  Call Extruder(264.21579)
  MoveL 9606 to (525.09, 528.57, 172) mm, rotated rx 180 ry 0 rz 160 deg; joints [9.282, 56.814, -9.011, -142.877, 54.137, 156.086]
  Call Extruder(269.11621)
  MoveL 9607 to (523.93, 529.55, 172) mm, rotated rx -180 ry 0 rz 160 deg; joints [9.42, 56.63, -8.662, -142.793, 54.323, 156.117]
  Set speed (17.5 mm/s)
  Call Extruder(272.14590)
  MoveL 9608 to (523.2, 530.13, 172) mm, rotated rx -180 ry 0 rz 160 deg; joints [9.503, 56.512, -8.44, -142.745, 54.44, 156.14]
  Set speed (17.5 mm/s)
  Call Extruder(276.64119)
  MoveL 9609 to (522.08, 530.96, 172) mm, rotated rx -180 ry 0 rz 160 deg; joints [9.623, 56.332, -8.101, -142.679, 54.616, 156.181]
  Set speed (17.5 mm/s)
  Call Extruder(279.35040)
  MoveL 9610 to (521.39, 531.44, 172) mm, rotated rx 180 ry 0 rz 160 deg; joints [9.693, 56.221, -7.89, -142.643, 54.723, 156.208]
  Set speed (17.5 mm/s)
  Call Extruder(281.76760)
  MoveL 9611 to (520.77, 531.85, 172) mm, rotated rx -180 ry 0 rz 160 deg; joints [9.755, 56.12, -7.7, -142.612, 54.819, 156.235]
  Set speed (17.5 mm/s)
  Call Extruder(284.79201)
  MoveL 9612 to (519.98, 532.36, 172) mm, rotated rx 180 ry 0 rz 160 deg; joints [9.831, 55.992, -7.459, -142.576, 54.939, 156.27]
  Set speed (17.5 mm/s)
  Call Extruder(286.82384)
  MoveL 9613 to (519.44, 532.68, 172) mm, rotated rx 180 ry 0 rz 160 deg; joints [9.881, 55.905, -7.294, -142.553, 55.021, 156.296]
  Set speed (17.5 mm/s)
  Call Extruder(289.33819)
  MoveL 9614 to (518.77, 533.08, 172) mm, rotated rx 180 ry 0 rz 160 deg; joints [9.941, 55.795, -7.088, -142.527, 55.122, 156.329]
  Set speed (17.5 mm/s)
  Call Extruder(291.88729)
  MoveL 9615 to (518.08, 533.46, 172) mm, rotated rx 180 ry 0 rz 160 deg; joints [10.001, 55.682, -6.875, -142.502, 55.225, 156.365]
  Call Extruder(294.64849)
  MoveL 9616 to (517.32, 533.86, 172) mm, rotated rx 180 ry 0 rz 160 deg; joints [10.064, 55.559, -6.642, -142.478, 55.337, 156.406]
  Set speed (17.5 mm/s)
  Call Extruder(299.60980)
  MoveL 9617 to (515.94, 534.53, 172) mm, rotated rx -180 ry 0 rz 160 deg; joints [10.173, 55.333, -6.215, -142.44, 55.54, 156.485]
  Set speed (17.5 mm/s)
  Call Extruder(304.71552)
  MoveL 9618 to (514.49, 535.16, 172) mm, rotated rx 180 ry 0 rz 160 deg; joints [10.28, 55.095, -5.766, -142.41, 55.75, 156.574]
  Set speed (17.5 mm/s)
  Call Extruder(309.41983)
  MoveL 9619 to (513.13, 535.69, 172) mm, rotated rx -180 ry 0 rz 160 deg; joints [10.373, 54.871, -5.344, -142.388, 55.944, 156.662]
  Call Extruder(314.52276)
  MoveL 9620 to (511.64, 536.2, 172) mm, rotated rx -180 ry 0 rz 160 deg; joints [10.468, 54.624, -4.879, -142.373, 56.154, 156.765]
  Set speed (17.5 mm/s)
  Call Extruder(319.40100)
  MoveL 9621 to (510.19, 536.64, 172) mm, rotated rx 180 ry 0 rz 160 deg; joints [10.553, 54.384, -4.427, -142.366, 56.356, 156.869]
  Set speed (17.5 mm/s)
  Call Extruder(324.41187)
  MoveL 9622 to (508.69, 537.02, 172) mm, rotated rx 180 ry 0 rz 160 deg; joints [10.633, 54.135, -3.957, -142.367, 56.562, 156.981]
  Set speed (17.5 mm/s)
  Call Extruder(329.43968)
  MoveL 9623 to (507.17, 537.35, 172) mm, rotated rx 180 ry 0 rz 160 deg; joints [10.707, 53.882, -3.479, -142.376, 56.768, 157.1]
  Set speed (17.5 mm/s)
  Call Extruder(334.69209)
  MoveL 9624 to (505.57, 537.62, 172) mm, rotated rx -180 ry 0 rz 160 deg; joints [10.777, 53.614, -2.975, -142.393, 56.983, 157.231]
  Call Extruder(339.62073)
  MoveL 9625 to (504.05, 537.81, 172) mm, rotated rx -180 ry 0 rz 160 deg; joints [10.835, 53.361, -2.498, -142.417, 57.183, 157.359]
  Set speed (17.5 mm/s)
  Call Extruder(344.69311)
  MoveL 9626 to (502.49, 537.95, 172) mm, rotated rx 180 ry 0 rz 160 deg; joints [10.889, 53.099, -2.004, -142.449, 57.387, 157.495]
  Call Extruder(349.77465)
  MoveL 9627 to (500.91, 538.02, 172) mm, rotated rx -180 ry 0 rz 160 deg; joints [10.934, 52.835, -1.506, -142.49, 57.59, 157.637]
  Set speed (17.5 mm/s)
  Call Extruder(354.61934)
  MoveL 9628 to (499.41, 538.02, 172) mm, rotated rx -180 ry 0 rz 160 deg; joints [10.971, 52.582, -1.03, -142.536, 57.781, 157.776]
  Set speed (10.0 mm/s)
  MoveL 9629 to (499.41, 538.02, 176) mm, rotated rx 180 ry 0 rz 160 deg; joints [10.971, 52.04, -0.954, -142.356, 57.412, 157.44]
  Set speed (120.0 mm/s)
  MoveL 9630 to (499.43, 537.08, 176) mm, rotated rx 180 ry 0 rz 160 deg; joints [10.855, 52.012, -0.902, -142.492, 57.387, 157.526]
  Set speed (17.6 mm/s)
  Call Extruder(359.63179)
  MoveL 9631 to (497.87, 537.03, 176) mm, rotated rx -180 ry 0 rz 160 deg; joints [10.885, 51.747, -0.406, -142.549, 57.581, 157.675]
  Call Extruder(364.52764)
  MoveL 9632 to (496.35, 536.91, 176) mm, rotated rx -180 ry 0 rz 160 deg; joints [10.906, 51.489, 0.078, -142.613, 57.768, 157.825]
  Call Extruder(369.33210)
  MoveL 9633 to (494.87, 536.73, 176) mm, rotated rx 180 ry 0 rz 160 deg; joints [10.92, 51.235, 0.552, -142.682, 57.949, 157.975]
  Set speed (17.6 mm/s)
  Call Extruder(374.09373)
  MoveL 9634 to (493.4, 536.49, 176) mm, rotated rx 180 ry 0 rz 160 deg; joints [10.925, 50.984, 1.022, -142.758, 58.125, 158.128]
  Call Extruder(378.49274)
  MoveL 9635 to (492.06, 536.23, 176) mm, rotated rx -180 ry 0 rz 160 deg; joints [10.925, 50.754, 1.453, -142.834, 58.284, 158.271]
  Set speed (17.6 mm/s)
  Call Extruder(381.55349)
  MoveL 9636 to (491.13, 536.01, 176) mm, rotated rx -180 ry 0 rz 160 deg; joints [10.92, 50.594, 1.751, -142.891, 58.393, 158.372]
  Call Extruder(383.93419)
  MoveL 9637 to (490.41, 535.83, 176) mm, rotated rx -180 ry 0 rz 160 deg; joints [10.914, 50.47, 1.983, -142.937, 58.477, 158.451]
  Set speed (17.6 mm/s)
  Call Extruder(388.87401)
  MoveL 9638 to (488.93, 535.4, 176) mm, rotated rx 180 ry 0 rz 160 deg; joints [10.896, 50.215, 2.46, -143.038, 58.648, 158.618]
  Set speed (17.6 mm/s)
  Call Extruder(393.64536)
  MoveL 9639 to (487.52, 534.93, 176) mm, rotated rx -180 ry 0 rz 160 deg; joints [10.871, 49.971, 2.916, -143.144, 58.808, 158.782]
  Set speed (17.6 mm/s)
  Call Extruder(398.69949)
  MoveL 9640 to (486.06, 534.37, 176) mm, rotated rx -180 ry 0 rz 160 deg; joints [10.835, 49.715, 3.395, -143.262, 58.973, 158.957]
  Set speed (17.6 mm/s)
  Call Extruder(403.34117)
  MoveL 9641 to (484.73, 533.8, 176) mm, rotated rx 180 ry 0 rz 160 deg; joints [10.795, 49.483, 3.828, -143.378, 59.121, 159.12]
  Set speed (17.6 mm/s)
  Call Extruder(407.92857)
  MoveL 9642 to (483.44, 533.18, 176) mm, rotated rx 180 ry 0 rz 160 deg; joints [10.748, 49.256, 4.251, -143.499, 59.262, 159.282]
  Set speed (17.6 mm/s)
  Call Extruder(411.24892)
  MoveL 9643 to (482.52, 532.71, 176) mm, rotated rx -180 ry 0 rz 160 deg; joints [10.71, 49.094, 4.553, -143.59, 59.361, 159.4]
  Set speed (17.6 mm/s)
  Call Extruder(415.20714)
  MoveL 9644 to (481.44, 532.11, 176) mm, rotated rx 180 ry 0 rz 160 deg; joints [10.659, 48.904, 4.908, -143.704, 59.476, 159.542]
  Set speed (17.6 mm/s)
  Call Extruder(417.70243)
  MoveL 9645 to (480.77, 531.71, 176) mm, rotated rx 180 ry 0 rz 160 deg; joints [10.624, 48.786, 5.129, -143.777, 59.546, 159.632]
  Set speed (17.6 mm/s)
  Call Extruder(420.49475)
  MoveL 9646 to (480.03, 531.25, 176) mm, rotated rx 180 ry 0 rz 160 deg; joints [10.583, 48.655, 5.374, -143.862, 59.624, 159.733]
  Call Extruder(425.15951)
  MoveL 9647 to (478.82, 530.45, 176) mm, rotated rx -180 ry 0 rz 160 deg; joints [10.508, 48.439, 5.776, -144.007, 59.749, 159.901]
  Set speed (17.6 mm/s)
  Call Extruder(427.37809)
  MoveL 9648 to (478.26, 530.05, 176) mm, rotated rx 180 ry 0 rz 160 deg; joints [10.469, 48.338, 5.964, -144.079, 59.806, 159.981]
  Set speed (17.6 mm/s)
  Call Extruder(430.26889)
  MoveL 9649 to (477.54, 529.51, 176) mm, rotated rx 180 ry 0 rz 160 deg; joints [10.417, 48.208, 6.207, -144.174, 59.88, 160.086]
  Set speed (17.6 mm/s)
  Call Extruder(432.68875)
  MoveL 9650 to (476.94, 529.05, 176) mm, rotated rx 180 ry 0 rz 160 deg; joints [10.371, 48.101, 6.406, -144.255, 59.939, 160.174]
  Set speed (17.6 mm/s)
  Call Extruder(437.16751)
  MoveL 9651 to (475.87, 528.16, 176) mm, rotated rx 180 ry 0 rz 160 deg; joints [10.281, 47.906, 6.769, -144.41, 60.045, 160.336]
  Set speed (17.6 mm/s)
  Call Extruder(439.64918)
  MoveL 9652 to (475.28, 527.65, 176) mm, rotated rx 180 ry 0 rz 160 deg; joints [10.228, 47.801, 6.967, -144.498, 60.102, 160.426]
  Set speed (17.6 mm/s)
  Call Extruder(443.32920)
  MoveL 9653 to (474.44, 526.87, 176) mm, rotated rx 180 ry 0 rz 160 deg; joints [10.147, 47.647, 7.254, -144.631, 60.183, 160.559]
  Set speed (17.6 mm/s)
  Call Extruder(448.58769)
  MoveL 9654 to (473.28, 525.72, 176) mm, rotated rx 180 ry 0 rz 160 deg; joints [10.022, 47.433, 7.652, -144.827, 60.293, 160.749]
  Set speed (17.6 mm/s)
  Call Extruder(452.04675)
  MoveL 9655 to (472.54, 524.93, 176) mm, rotated rx -180 ry 0 rz 160 deg; joints [9.936, 47.297, 7.905, -144.96, 60.36, 160.873]
  Set speed (17.6 mm/s)
  Call Extruder(457.05308)
  MoveL 9656 to (471.52, 523.76, 176) mm, rotated rx 180 ry 0 rz 160 deg; joints [9.804, 47.106, 8.261, -145.157, 60.452, 161.053]
  Set speed (17.6 mm/s)
  Call Extruder(459.37149)
  MoveL 9657 to (471.06, 523.2, 176) mm, rotated rx -180 ry 0 rz 160 deg; joints [9.74, 47.021, 8.42, -145.25, 60.492, 161.135]
  Set speed (17.6 mm/s)
  Call Extruder(463.94801)
  MoveL 9658 to (470.19, 522.07, 176) mm, rotated rx 180 ry 0 rz 160 deg; joints [9.61, 46.856, 8.727, -145.437, 60.567, 161.297]
  Set speed (17.6 mm/s)
  Call Extruder(466.71586)
  MoveL 9659 to (469.69, 521.37, 176) mm, rotated rx 180 ry 0 rz 160 deg; joints [9.528, 46.76, 8.906, -145.552, 60.61, 161.395]
  Set speed (17.6 mm/s)
  Call Extruder(469.23384)
  MoveL 9660 to (469.24, 520.72, 176) mm, rotated rx 180 ry 0 rz 160 deg; joints [9.453, 46.674, 9.065, -145.658, 60.646, 161.483]
  Set speed (17.6 mm/s)
  Call Extruder(471.45627)
  MoveL 9661 to (468.86, 520.14, 176) mm, rotated rx -180 ry 0 rz 160 deg; joints [9.384, 46.601, 9.202, -145.753, 60.677, 161.561]
  Set speed (17.6 mm/s)
  Call Extruder(474.03432)
  MoveL 9662 to (468.43, 519.47, 176) mm, rotated rx 180 ry 0 rz 160 deg; joints [9.302, 46.518, 9.356, -145.864, 60.71, 161.65]
  Set speed (17.6 mm/s)
  Call Extruder(478.56657)
  MoveL 9663 to (467.71, 518.25, 176) mm, rotated rx 180 ry 0 rz 160 deg; joints [9.156, 46.377, 9.619, -146.062, 60.765, 161.806]
  Set speed (17.6 mm/s)
  Call Extruder(481.44140)
  MoveL 9664 to (467.28, 517.47, 176) mm, rotated rx 180 ry 0 rz 160 deg; joints [9.06, 46.291, 9.778, -146.189, 60.796, 161.904]
  Set speed (17.6 mm/s)
  Call Extruder(483.77425)
  MoveL 9665 to (466.95, 516.82, 176) mm, rotated rx 180 ry 0 rz 160 deg; joints [8.981, 46.224, 9.903, -146.293, 60.82, 161.983]
  Set speed (17.6 mm/s)
  Call Extruder(486.19823)
  MoveL 9666 to (466.61, 516.15, 176) mm, rotated rx 180 ry 0 rz 160 deg; joints [8.897, 46.157, 10.029, -146.402, 60.842, 162.065]
  Set speed (17.6 mm/s)
  Call Extruder(491.16134)
  MoveL 9667 to (465.97, 514.74, 176) mm, rotated rx 180 ry 0 rz 160 deg; joints [8.721, 46.025, 10.275, -146.629, 60.883, 162.23]
  Set speed (17.6 mm/s)
  Call Extruder(495.80865)
  MoveL 9668 to (465.42, 513.4, 176) mm, rotated rx -180 ry 0 rz 160 deg; joints [8.551, 45.91, 10.488, -146.844, 60.914, 162.381]
  Set speed (17.6 mm/s)
  Call Extruder(497.97951)
  MoveL 9669 to (465.18, 512.77, 176) mm, rotated rx 180 ry 0 rz 160 deg; joints [8.471, 45.859, 10.583, -146.945, 60.926, 162.452]
  Set speed (17.6 mm/s)
  Call Extruder(500.75579)
  MoveL 9670 to (464.89, 511.95, 176) mm, rotated rx 180 ry 0 rz 160 deg; joints [8.366, 45.797, 10.699, -147.076, 60.94, 162.54]
  Set speed (17.6 mm/s)
  Call Extruder(505.52361)
  MoveL 9671 to (464.44, 510.54, 176) mm, rotated rx 180 ry 0 rz 160 deg; joints [8.184, 45.696, 10.885, -147.301, 60.958, 162.691]
  Set speed (17.6 mm/s)
  Call Extruder(510.42166)
  MoveL 9672 to (464.04, 509.07, 176) mm, rotated rx 180 ry 0 rz 160 deg; joints [7.991, 45.603, 11.058, -147.535, 60.968, 162.842]
  Set speed (17.6 mm/s)
  Call Extruder(512.49718)
  MoveL 9673 to (463.89, 508.44, 176) mm, rotated rx -180 ry 0 rz 160 deg; joints [7.909, 45.567, 11.126, -147.635, 60.97, 162.905]
  Set speed (17.5 mm/s)
  Call Extruder(515.99585)
  MoveL 9674 to (463.65, 507.38, 176) mm, rotated rx 180 ry 0 rz 160 deg; joints [7.769, 45.509, 11.234, -147.803, 60.971, 163.01]
  Set speed (17.6 mm/s)
  Call Extruder(520.41209)
  MoveL 9675 to (463.4, 506.03, 176) mm, rotated rx 180 ry 0 rz 160 deg; joints [7.589, 45.443, 11.356, -148.016, 60.967, 163.139]
  Set speed (17.6 mm/s)
  Call Extruder(525.27094)
  MoveL 9676 to (463.19, 504.53, 176) mm, rotated rx 180 ry 0 rz 160 deg; joints [7.388, 45.381, 11.472, -148.251, 60.954, 163.278]
  Set speed (17.6 mm/s)
  Call Extruder(530.14625)
  MoveL 9677 to (463.04, 503.02, 176) mm, rotated rx 180 ry 0 rz 160 deg; joints [7.184, 45.328, 11.57, -148.488, 60.935, 163.414]
  Set speed (17.6 mm/s)
  Call Extruder(534.85806)
  MoveL 9678 to (462.95, 501.55, 176) mm, rotated rx -180 ry 0 rz 160 deg; joints [6.985, 45.287, 11.647, -148.716, 60.908, 163.541]
  Call Extruder(540.27493)
  MoveL 9679 to (462.91, 499.87, 176) mm, rotated rx -180 ry 0 rz 160 deg; joints [6.755, 45.251, 11.713, -148.978, 60.87, 163.683]
  Call Extruder(544.26304)
  MoveL 9680 to (462.94, 498.62, 176) mm, rotated rx -180 ry 0 rz 160 deg; joints [6.584, 45.233, 11.747, -149.171, 60.835, 163.783]
  Set speed (17.6 mm/s)
  Call Extruder(548.49885)
  MoveL 9681 to (463.01, 497.31, 176) mm, rotated rx -180 ry 0 rz 160 deg; joints [6.402, 45.221, 11.769, -149.374, 60.793, 163.887]
  Set speed (17.6 mm/s)
  Call Extruder(552.94201)
  MoveL 9682 to (463.14, 495.93, 176) mm, rotated rx 180 ry 0 rz 160 deg; joints [6.211, 45.217, 11.777, -149.585, 60.744, 163.992]
  Set speed (17.6 mm/s)
  Call Extruder(557.33534)
  MoveL 9683 to (463.31, 494.57, 176) mm, rotated rx -180 ry 0 rz 160 deg; joints [6.022, 45.222, 11.768, -149.792, 60.688, 164.091]
  Set speed (17.6 mm/s)
  Call Extruder(561.79803)
  MoveL 9684 to (463.54, 493.2, 176) mm, rotated rx -180 ry 0 rz 160 deg; joints [5.831, 45.235, 11.744, -150, 60.626, 164.188]
  Call Extruder(566.04683)
  MoveL 9685 to (463.81, 491.9, 176) mm, rotated rx 180 ry 0 rz 160 deg; joints [5.649, 45.255, 11.705, -150.196, 60.561, 164.277]
  Set speed (17.6 mm/s)
  Call Extruder(570.30848)
  MoveL 9686 to (464.12, 490.61, 176) mm, rotated rx 180 ry 0 rz 160 deg; joints [5.468, 45.284, 11.652, -150.39, 60.491, 164.361]
  Set speed (17.6 mm/s)
  Call Extruder(574.80817)
  MoveL 9687 to (464.5, 489.27, 176) mm, rotated rx 180 ry 0 rz 160 deg; joints [5.278, 45.323, 11.58, -150.591, 60.411, 164.446]
  Call Extruder(579.25382)
  MoveL 9688 to (464.93, 487.95, 176) mm, rotated rx 180 ry 0 rz 160 deg; joints [5.092, 45.369, 11.494, -150.786, 60.326, 164.526]
  Set speed (17.6 mm/s)
  Call Extruder(583.67764)
  MoveL 9689 to (465.4, 486.65, 176) mm, rotated rx -180 ry 0 rz 160 deg; joints [4.908, 45.424, 11.392, -150.977, 60.236, 164.6]
  Set speed (17.6 mm/s)
  Call Extruder(587.21852)
  MoveL 9690 to (465.81, 485.63, 176) mm, rotated rx -180 ry 0 rz 160 deg; joints [4.763, 45.473, 11.3, -151.126, 60.161, 164.657]
  Set speed (17.6 mm/s)
  Call Extruder(592.49741)
  MoveL 9691 to (466.48, 484.13, 176) mm, rotated rx 180 ry 0 rz 160 deg; joints [4.55, 45.557, 11.144, -151.343, 60.041, 164.735]
  Set speed (17.6 mm/s)
  Call Extruder(596.74590)
  MoveL 9692 to (467.07, 482.95, 176) mm, rotated rx -180 ry 0 rz 160 deg; joints [4.382, 45.633, 11.003, -151.512, 59.94, 164.793]
  Set speed (17.6 mm/s)
  Call Extruder(601.02028)
  MoveL 9693 to (467.7, 481.77, 176) mm, rotated rx -180 ry 0 rz 160 deg; joints [4.215, 45.717, 10.847, -151.679, 59.833, 164.846]
  Set speed (17.6 mm/s)
  Call Extruder(605.60569)
  MoveL 9694 to (468.42, 480.55, 176) mm, rotated rx -180 ry 0 rz 160 deg; joints [4.04, 45.814, 10.665, -151.851, 59.713, 164.899]
  Call Extruder(609.80250)
  MoveL 9695 to (469.13, 479.45, 176) mm, rotated rx 180 ry 0 rz 160 deg; joints [3.883, 45.912, 10.485, -152.003, 59.599, 164.942]
  Set speed (17.6 mm/s)
  Call Extruder(614.16058)
  MoveL 9696 to (469.9, 478.33, 176) mm, rotated rx -180 ry 0 rz 160 deg; joints [3.724, 46.019, 10.285, -152.156, 59.476, 164.982]
  Set speed (17.6 mm/s)
  Call Extruder(618.80144)
  MoveL 9697 to (470.77, 477.17, 176) mm, rotated rx -180 ry 0 rz 160 deg; joints [3.56, 46.142, 10.056, -152.312, 59.34, 165.019]
  Set speed (17.6 mm/s)
  Call Extruder(623.02775)
  MoveL 9698 to (471.6, 476.15, 176) mm, rotated rx -180 ry 0 rz 160 deg; joints [3.414, 46.261, 9.835, -152.447, 59.211, 165.047]
  Set speed (17.6 mm/s)
  Call Extruder(627.38380)
  MoveL 9699 to (472.49, 475.13, 176) mm, rotated rx -180 ry 0 rz 160 deg; joints [3.268, 46.39, 9.595, -152.581, 59.075, 165.072]
  Set speed (17.6 mm/s)
  Call Extruder(631.78306)
  MoveL 9700 to (473.43, 474.13, 176) mm, rotated rx 180 ry 0 rz 160 deg; joints [3.126, 46.527, 9.34, -152.708, 58.934, 165.091]
  Set speed (17.6 mm/s)
  Call Extruder(636.24796)
  MoveL 9701 to (474.42, 473.15, 176) mm, rotated rx 180 ry 0 rz 160 deg; joints [2.987, 46.673, 9.068, -152.831, 58.786, 165.105]
  Set speed (17.6 mm/s)
  Call Extruder(640.67109)
  MoveL 9702 to (475.43, 472.22, 176) mm, rotated rx -180 ry 0 rz 160 deg; joints [2.854, 46.824, 8.786, -152.944, 58.636, 165.113]
  Set speed (17.6 mm/s)
  Call Extruder(644.84265)
  MoveL 9703 to (476.42, 471.37, 176) mm, rotated rx -180 ry 0 rz 160 deg; joints [2.734, 46.973, 8.509, -153.045, 58.491, 165.116]
  Call Extruder(649.39966)
  MoveL 9704 to (477.53, 470.49, 176) mm, rotated rx -180 ry 0 rz 160 deg; joints [2.609, 47.141, 8.195, -153.146, 58.329, 165.113]
  Call Extruder(653.88093)
  MoveL 9705 to (478.66, 469.67, 176) mm, rotated rx -180 ry 0 rz 160 deg; joints [2.492, 47.313, 7.876, -153.238, 58.167, 165.104]
  Set speed (17.6 mm/s)
  Call Extruder(658.06133)
  MoveL 9706 to (479.74, 468.94, 176) mm, rotated rx 180 ry 0 rz 160 deg; joints [2.389, 47.478, 7.567, -153.316, 58.012, 165.091]
  Call Extruder(662.47412)
  MoveL 9707 to (480.9, 468.21, 176) mm, rotated rx -180 ry 0 rz 160 deg; joints [2.285, 47.658, 7.232, -153.39, 57.847, 165.071]
  Call Extruder(667.00965)
  MoveL 9708 to (482.13, 467.5, 176) mm, rotated rx 180 ry 0 rz 160 deg; joints [2.185, 47.849, 6.877, -153.458, 57.674, 165.045]
  Set speed (17.6 mm/s)
  Call Extruder(671.23016)
  MoveL 9709 to (483.29, 466.89, 176) mm, rotated rx 180 ry 0 rz 160 deg; joints [2.098, 48.031, 6.538, -153.513, 57.511, 165.015]
  Set speed (17.6 mm/s)
  Call Extruder(675.73847)
  MoveL 9710 to (484.56, 466.28, 176) mm, rotated rx 180 ry 0 rz 160 deg; joints [2.012, 48.23, 6.166, -153.563, 57.334, 164.978]
  Set speed (17.6 mm/s)
  Call Extruder(680.17652)
  MoveL 9711 to (485.82, 465.73, 176) mm, rotated rx 180 ry 0 rz 160 deg; joints [1.933, 48.43, 5.792, -153.603, 57.158, 164.935]
  Set speed (17.6 mm/s)
  Call Extruder(684.45952)
  MoveL 9712 to (487.06, 465.24, 176) mm, rotated rx -180 ry 0 rz 160 deg; joints [1.864, 48.628, 5.424, -153.634, 56.987, 164.888]
  Call Extruder(688.93282)
  MoveL 9713 to (488.38, 464.78, 176) mm, rotated rx -180 ry 0 rz 160 deg; joints [1.798, 48.838, 5.031, -153.657, 56.806, 164.833]
  Set speed (17.6 mm/s)
  Call Extruder(693.16871)
  MoveL 9714 to (489.64, 464.39, 176) mm, rotated rx -180 ry 0 rz 160 deg; joints [1.742, 49.041, 4.653, -153.671, 56.634, 164.775]
  Call Extruder(697.69921)
  MoveL 9715 to (491, 464.02, 176) mm, rotated rx 180 ry 0 rz 160 deg; joints [1.688, 49.261, 4.242, -153.677, 56.449, 164.707]
  Set speed (17.6 mm/s)
  Call Extruder(701.99485)
  MoveL 9716 to (492.3, 463.72, 176) mm, rotated rx -180 ry 0 rz 160 deg; joints [1.645, 49.473, 3.846, -153.673, 56.273, 164.638]
  Set speed (17.6 mm/s)
  Call Extruder(706.30892)
  MoveL 9717 to (493.62, 463.47, 176) mm, rotated rx -180 ry 0 rz 160 deg; joints [1.607, 49.689, 3.443, -153.662, 56.095, 164.562]
  Set speed (17.6 mm/s)
  Call Extruder(710.54344)
  MoveL 9718 to (494.93, 463.26, 176) mm, rotated rx 180 ry 0 rz 160 deg; joints [1.575, 49.902, 3.044, -153.642, 55.92, 164.483]
  Set speed (17.6 mm/s)
  Call Extruder(715.19540)
  MoveL 9719 to (496.37, 463.09, 176) mm, rotated rx -180 ry 0 rz 160 deg; joints [1.549, 50.14, 2.6, -153.611, 55.728, 164.39]
  Set speed (17.6 mm/s)
  Call Extruder(719.45807)
  MoveL 9720 to (497.69, 462.98, 176) mm, rotated rx -180 ry 0 rz 160 deg; joints [1.53, 50.36, 2.189, -153.574, 55.552, 164.299]
  Set speed (17.6 mm/s)
  Call Extruder(723.99441)
  MoveL 9721 to (499.1, 462.92, 176) mm, rotated rx 180 ry 0 rz 160 deg; joints [1.518, 50.595, 1.749, -153.526, 55.366, 164.196]
  Call Extruder(728.30512)
  MoveL 9722 to (500.45, 462.92, 176) mm, rotated rx 180 ry 0 rz 160 deg; joints [1.512, 50.821, 1.327, -153.472, 55.189, 164.094]
  Call Extruder(732.77186)
  MoveL 9723 to (501.84, 462.96, 176) mm, rotated rx 180 ry 0 rz 160 deg; joints [1.513, 51.055, 0.889, -153.408, 55.006, 163.982]
  Set speed (17.6 mm/s)
  Call Extruder(737.07059)
  MoveL 9724 to (503.17, 463.05, 176) mm, rotated rx -180 ry 0 rz 160 deg; joints [1.52, 51.282, 0.465, -153.338, 54.832, 163.869]
  Call Extruder(741.53196)
  MoveL 9725 to (504.55, 463.19, 176) mm, rotated rx 180 ry 0 rz 160 deg; joints [1.534, 51.517, 0.024, -153.256, 54.652, 163.747]
  Set speed (17.6 mm/s)
  Call Extruder(745.77816)
  MoveL 9726 to (505.86, 463.38, 176) mm, rotated rx 180 ry 0 rz 160 deg; joints [1.553, 51.742, -0.396, -153.171, 54.483, 163.626]
  Set speed (17.6 mm/s)
  Call Extruder(750.20388)
  MoveL 9727 to (507.22, 463.62, 176) mm, rotated rx -180 ry 0 rz 160 deg; joints [1.579, 51.976, -0.833, -153.074, 54.309, 163.495]
  Set speed (17.6 mm/s)
  Call Extruder(754.02906)
  MoveL 9728 to (508.38, 463.87, 176) mm, rotated rx -180 ry 0 rz 160 deg; joints [1.606, 52.177, -1.211, -152.985, 54.16, 163.378]
  Call Extruder(758.99083)
  MoveL 9729 to (509.88, 464.25, 176) mm, rotated rx 180 ry 0 rz 160 deg; joints [1.648, 52.438, -1.699, -152.86, 53.969, 163.221]
  Set speed (17.6 mm/s)
  Call Extruder(763.35975)
  MoveL 9730 to (511.18, 464.64, 176) mm, rotated rx 180 ry 0 rz 160 deg; joints [1.691, 52.667, -2.128, -152.742, 53.804, 163.077]
  Set speed (17.6 mm/s)
  Call Extruder(767.84305)
  MoveL 9731 to (512.51, 465.09, 176) mm, rotated rx -180 ry 0 rz 160 deg; joints [1.742, 52.901, -2.566, -152.613, 53.638, 162.926]
  Set speed (17.6 mm/s)
  Call Extruder(772.13439)
  MoveL 9732 to (513.76, 465.56, 176) mm, rotated rx 180 ry 0 rz 160 deg; joints [1.795, 53.123, -2.982, -152.484, 53.481, 162.777]
  Call Extruder(776.60866)
  MoveL 9733 to (515.04, 466.1, 176) mm, rotated rx -180 ry 0 rz 160 deg; joints [1.857, 53.353, -3.412, -152.341, 53.322, 162.617]
  Call Extruder(780.94194)
  MoveL 9734 to (516.27, 466.67, 176) mm, rotated rx -180 ry 0 rz 160 deg; joints [1.922, 53.573, -3.825, -152.197, 53.171, 162.459]
  Call Extruder(785.32245)
  MoveL 9735 to (517.48, 467.29, 176) mm, rotated rx -180 ry 0 rz 160 deg; joints [1.994, 53.793, -4.238, -152.044, 53.022, 162.295]
  Set speed (17.6 mm/s)
  Call Extruder(789.75529)
  MoveL 9736 to (518.69, 467.96, 176) mm, rotated rx -180 ry 0 rz 160 deg; joints [2.071, 54.013, -4.651, -151.884, 52.876, 162.127]
  Set speed (17.6 mm/s)
  Call Extruder(794.04371)
  MoveL 9737 to (519.83, 468.66, 176) mm, rotated rx -180 ry 0 rz 160 deg; joints [2.15, 54.223, -5.044, -151.723, 52.739, 161.96]
  Call Extruder(798.51529)
  MoveL 9738 to (520.99, 469.43, 176) mm, rotated rx 180 ry 0 rz 160 deg; joints [2.239, 54.439, -5.448, -151.549, 52.601, 161.784]
  Set speed (17.6 mm/s)
  Call Extruder(802.75656)
  MoveL 9739 to (522.07, 470.19, 176) mm, rotated rx 180 ry 0 rz 160 deg; joints [2.327, 54.639, -5.824, -151.38, 52.474, 161.614]
  Set speed (17.6 mm/s)
  Call Extruder(807.05697)
  MoveL 9740 to (523.13, 471.01, 176) mm, rotated rx 180 ry 0 rz 160 deg; joints [2.42, 54.839, -6.198, -151.203, 52.35, 161.44]
  Set speed (17.6 mm/s)
  Call Extruder(811.62276)
  MoveL 9741 to (524.22, 471.92, 176) mm, rotated rx -180 ry 0 rz 160 deg; joints [2.524, 55.047, -6.588, -151.011, 52.224, 161.252]
  Call Extruder(816.01638)
  MoveL 9742 to (525.24, 472.83, 176) mm, rotated rx 180 ry 0 rz 160 deg; joints [2.629, 55.241, -6.954, -150.821, 52.109, 161.07]
  Set speed (17.6 mm/s)
  Call Extruder(820.27521)
  MoveL 9743 to (526.2, 473.75, 176) mm, rotated rx -180 ry 0 rz 160 deg; joints [2.734, 55.426, -7.3, -150.633, 52.002, 160.893]
  Set speed (17.6 mm/s)
  Call Extruder(822.37466)
  MoveL 9744 to (526.66, 474.22, 176) mm, rotated rx -180 ry 0 rz 160 deg; joints [2.787, 55.515, -7.467, -150.539, 51.952, 160.804]
  Set speed (17.6 mm/s)
  Call Extruder(824.99208)
  MoveL 9745 to (527.22, 474.81, 176) mm, rotated rx -180 ry 0 rz 160 deg; joints [2.855, 55.624, -7.672, -150.42, 51.891, 160.694]
  Set speed (17.6 mm/s)
  Call Extruder(827.30124)
  MoveL 9746 to (527.7, 475.34, 176) mm, rotated rx 180 ry 0 rz 160 deg; joints [2.916, 55.719, -7.85, -150.315, 51.838, 160.597]
  Set speed (17.6 mm/s)
  Call Extruder(830.24036)
  MoveL 9747 to (528.3, 476.03, 176) mm, rotated rx -180 ry 0 rz 160 deg; joints [2.995, 55.838, -8.073, -150.18, 51.774, 160.472]
  Set speed (17.6 mm/s)
  Call Extruder(834.48297)
  MoveL 9748 to (529.14, 477.06, 176) mm, rotated rx 180 ry 0 rz 160 deg; joints [3.112, 56.005, -8.386, -149.982, 51.687, 160.293]
  Set speed (17.6 mm/s)
  Call Extruder(836.98069)
  MoveL 9749 to (529.61, 477.67, 176) mm, rotated rx -180 ry 0 rz 160 deg; joints [3.183, 56.1, -8.565, -149.864, 51.638, 160.187]
  Set speed (17.6 mm/s)
  Call Extruder(839.85041)
  MoveL 9750 to (530.14, 478.39, 176) mm, rotated rx -180 ry 0 rz 160 deg; joints [3.265, 56.208, -8.766, -149.728, 51.585, 160.065]
  Set speed (17.6 mm/s)
  Call Extruder(844.17741)
  MoveL 9751 to (530.91, 479.5, 176) mm, rotated rx 180 ry 0 rz 160 deg; joints [3.392, 56.364, -9.061, -149.521, 51.51, 159.882]
  Call Extruder(846.78175)
  MoveL 9752 to (531.35, 480.18, 176) mm, rotated rx -180 ry 0 rz 160 deg; joints [3.47, 56.455, -9.231, -149.395, 51.468, 159.772]
  Set speed (17.6 mm/s)
  Call Extruder(849.61570)
  MoveL 9753 to (531.81, 480.94, 176) mm, rotated rx 180 ry 0 rz 160 deg; joints [3.556, 56.552, -9.413, -149.257, 51.425, 159.652]
  Set speed (17.6 mm/s)
  Call Extruder(851.57073)
  MoveL 9754 to (532.12, 481.46, 176) mm, rotated rx -180 ry 0 rz 160 deg; joints [3.616, 56.617, -9.535, -149.162, 51.397, 159.57]
  Set speed (17.6 mm/s)
  Call Extruder(854.08931)
  MoveL 9755 to (532.51, 482.15, 176) mm, rotated rx -180 ry 0 rz 160 deg; joints [3.694, 56.698, -9.688, -149.039, 51.363, 159.465]
  Set speed (17.6 mm/s)
  Call Extruder(858.93666)
  MoveL 9756 to (533.21, 483.48, 176) mm, rotated rx -180 ry 0 rz 160 deg; joints [3.847, 56.849, -9.97, -148.801, 51.304, 159.263]
  Call Extruder(861.53872)
  MoveL 9757 to (533.56, 484.21, 176) mm, rotated rx 180 ry 0 rz 160 deg; joints [3.93, 56.926, -10.116, -148.673, 51.275, 159.155]
  Set speed (17.6 mm/s)
  Call Extruder(864.10850)
  MoveL 9758 to (533.89, 484.94, 176) mm, rotated rx 180 ry 0 rz 160 deg; joints [4.013, 56.999, -10.253, -148.547, 51.25, 159.05]
  Set speed (17.6 mm/s)
  Call Extruder(869.08673)
  MoveL 9759 to (534.49, 486.37, 176) mm, rotated rx -180 ry 0 rz 160 deg; joints [4.177, 57.134, -10.506, -148.301, 51.208, 158.848]
  Set speed (17.6 mm/s)
  Call Extruder(873.77970)
  MoveL 9760 to (535, 487.74, 176) mm, rotated rx 180 ry 0 rz 160 deg; joints [4.333, 57.252, -10.728, -148.07, 51.177, 158.66]
  Set speed (17.6 mm/s)
  Call Extruder(878.73492)
  MoveL 9761 to (535.48, 489.21, 176) mm, rotated rx -180 ry 0 rz 160 deg; joints [4.502, 57.366, -10.942, -147.826, 51.153, 158.466]
  Set speed (17.6 mm/s)
  Call Extruder(883.68251)
  MoveL 9762 to (535.9, 490.69, 176) mm, rotated rx -180 ry 0 rz 160 deg; joints [4.672, 57.47, -11.138, -147.583, 51.138, 158.276]
  Set speed (17.6 mm/s)
  Call Extruder(888.45640)
  MoveL 9763 to (536.24, 492.14, 176) mm, rotated rx 180 ry 0 rz 160 deg; joints [4.838, 57.56, -11.307, -147.351, 51.134, 158.097]
  Set speed (17.6 mm/s)
  Call Extruder(893.38970)
  MoveL 9764 to (536.54, 493.65, 176) mm, rotated rx 180 ry 0 rz 160 deg; joints [5.012, 57.643, -11.462, -147.112, 51.138, 157.916]
  Set speed (17.6 mm/s)
  Call Extruder(898.26246)
  MoveL 9765 to (536.77, 495.15, 176) mm, rotated rx 180 ry 0 rz 160 deg; joints [5.185, 57.714, -11.596, -146.879, 51.151, 157.744]
  Set speed (17.6 mm/s)
  Call Extruder(903.21913)
  MoveL 9766 to (536.94, 496.68, 176) mm, rotated rx -180 ry 0 rz 160 deg; joints [5.362, 57.775, -11.709, -146.645, 51.173, 157.574]
  Set speed (17.6 mm/s)
  Call Extruder(907.99971)
  MoveL 9767 to (537.04, 498.17, 176) mm, rotated rx 180 ry 0 rz 160 deg; joints [5.535, 57.823, -11.8, -146.422, 51.204, 157.416]
  Call Extruder(912.87314)
  MoveL 9768 to (537.09, 499.69, 176) mm, rotated rx 180 ry 0 rz 160 deg; joints [5.711, 57.861, -11.871, -146.198, 51.245, 157.261]
  Set speed (17.6 mm/s)
  Call Extruder(917.63353)
  MoveL 9769 to (537.07, 501.17, 176) mm, rotated rx -180 ry 0 rz 160 deg; joints [5.884, 57.886, -11.919, -145.983, 51.293, 157.117]
  Set speed (17.6 mm/s)
  Call Extruder(922.58395)
  MoveL 9770 to (536.99, 502.71, 176) mm, rotated rx 180 ry 0 rz 160 deg; joints [6.065, 57.902, -11.949, -145.764, 51.352, 156.974]
  Set speed (17.6 mm/s)
  Call Extruder(927.38395)
  MoveL 9771 to (536.85, 504.2, 176) mm, rotated rx 180 ry 0 rz 160 deg; joints [6.24, 57.906, -11.956, -145.556, 51.418, 156.843]
  Set speed (17.6 mm/s)
  Call Extruder(932.43605)
  MoveL 9772 to (536.64, 505.76, 176) mm, rotated rx 180 ry 0 rz 160 deg; joints [6.425, 57.899, -11.943, -145.342, 51.496, 156.712]
  Set speed (17.6 mm/s)
  Call Extruder(937.20078)
  MoveL 9773 to (536.38, 507.22, 176) mm, rotated rx 180 ry 0 rz 160 deg; joints [6.598, 57.881, -11.909, -145.146, 51.577, 156.597]
  Set speed (17.6 mm/s)
  Call Extruder(942.26009)
  MoveL 9774 to (536.04, 508.76, 176) mm, rotated rx -180 ry 0 rz 160 deg; joints [6.782, 57.85, -11.851, -144.943, 51.673, 156.483]
  Set speed (17.6 mm/s)
  Call Extruder(946.79489)
  MoveL 9775 to (535.68, 510.13, 176) mm, rotated rx 180 ry 0 rz 160 deg; joints [6.946, 57.811, -11.778, -144.767, 51.766, 156.39]
  Set speed (17.6 mm/s)
  Call Extruder(951.84402)
  MoveL 9776 to (535.22, 511.63, 176) mm, rotated rx 180 ry 0 rz 160 deg; joints [7.128, 57.758, -11.678, -144.576, 51.878, 156.293]
  Set speed (17.6 mm/s)
  Call Extruder(956.49417)
  MoveL 9777 to (534.74, 513, 176) mm, rotated rx -180 ry 0 rz 160 deg; joints [7.294, 57.698, -11.566, -144.407, 51.987, 156.213]
  Set speed (17.6 mm/s)
  Call Extruder(961.72313)
  MoveL 9778 to (534.13, 514.51, 176) mm, rotated rx -180 ry 0 rz 160 deg; joints [7.48, 57.619, -11.417, -144.224, 52.119, 156.132]
  Set speed (17.6 mm/s)
  Call Extruder(966.32666)
  MoveL 9779 to (533.55, 515.82, 176) mm, rotated rx -180 ry 0 rz 160 deg; joints [7.641, 57.539, -11.267, -144.068, 52.241, 156.069]
  Set speed (17.6 mm/s)
  Call Extruder(971.09422)
  MoveL 9780 to (532.88, 517.15, 176) mm, rotated rx -180 ry 0 rz 160 deg; joints [7.807, 57.447, -11.093, -143.914, 52.374, 156.013]
  Set speed (17.6 mm/s)
  Call Extruder(973.39101)
  MoveL 9781 to (532.55, 517.78, 176) mm, rotated rx 180 ry 0 rz 160 deg; joints [7.886, 57.399, -11.003, -143.842, 52.44, 155.989]
  Set speed (17.6 mm/s)
  Call Extruder(978.17343)
  MoveL 9782 to (531.81, 519.08, 176) mm, rotated rx 180 ry 0 rz 160 deg; joints [8.049, 57.291, -10.801, -143.697, 52.583, 155.945]
  Set speed (17.6 mm/s)
  Call Extruder(980.72077)
  MoveL 9783 to (531.39, 519.75, 176) mm, rotated rx -180 ry 0 rz 160 deg; joints [8.135, 57.23, -10.686, -143.623, 52.661, 155.925]
  Call Extruder(983.04991)
  MoveL 9784 to (531, 520.36, 176) mm, rotated rx -180 ry 0 rz 160 deg; joints [8.213, 57.171, -10.576, -143.557, 52.734, 155.909]
  Call Extruder(985.50952)
  MoveL 9785 to (530.57, 521, 176) mm, rotated rx 180 ry 0 rz 160 deg; joints [8.294, 57.107, -10.456, -143.489, 52.813, 155.895]
  Set speed (17.6 mm/s)
  Call Extruder(988.90632)
  MoveL 9786 to (529.96, 521.86, 176) mm, rotated rx -180 ry 0 rz 160 deg; joints [8.406, 57.016, -10.283, -143.397, 52.923, 155.878]
  Call Extruder(993.15514)
  MoveL 9787 to (529.16, 522.92, 176) mm, rotated rx 180 ry 0 rz 160 deg; joints [8.543, 56.893, -10.054, -143.288, 53.065, 155.863]
  Set speed (17.6 mm/s)
  Call Extruder(997.65358)
  MoveL 9788 to (528.27, 524, 176) mm, rotated rx 180 ry 0 rz 160 deg; joints [8.686, 56.756, -9.797, -143.179, 53.22, 155.856]
  Set speed (17.6 mm/s)
  Call Extruder(1000.12214)
  MoveL 9789 to (527.77, 524.58, 176) mm, rotated rx -180 ry 0 rz 160 deg; joints [8.763, 56.678, -9.65, -143.122, 53.306, 155.854]
  Set speed (17.6 mm/s)
  Call Extruder(1002.54011)
  MoveL 9790 to (527.26, 525.14, 176) mm, rotated rx -180 ry 0 rz 160 deg; joints [8.838, 56.6, -9.502, -143.068, 53.392, 155.855]
  Set speed (17.6 mm/s)
  Call Extruder(1005.23711)
  MoveL 9791 to (526.69, 525.75, 176) mm, rotated rx 180 ry 0 rz 160 deg; joints [8.921, 56.509, -9.333, -143.01, 53.489, 155.859]
  Set speed (17.6 mm/s)
  Call Extruder(1010.28345)
  MoveL 9792 to (525.57, 526.86, 176) mm, rotated rx 180 ry 0 rz 160 deg; joints [9.072, 56.333, -9.003, -142.907, 53.674, 155.873]
  Set speed (17.6 mm/s)
  Call Extruder(1012.60786)
  MoveL 9793 to (525.04, 527.35, 176) mm, rotated rx -180 ry 0 rz 160 deg; joints [9.14, 56.249, -8.844, -142.863, 53.761, 155.882]
  Set speed (17.6 mm/s)
  Call Extruder(1017.57129)
  MoveL 9794 to (523.88, 528.38, 176) mm, rotated rx 180 ry 0 rz 160 deg; joints [9.282, 56.064, -8.497, -142.773, 53.949, 155.909]
  Set speed (17.6 mm/s)
  Call Extruder(1020.03229)
  MoveL 9795 to (523.29, 528.86, 176) mm, rotated rx -180 ry 0 rz 160 deg; joints [9.351, 55.969, -8.319, -142.732, 54.043, 155.925]
  Set speed (17.6 mm/s)
  Call Extruder(1024.71071)
  MoveL 9796 to (522.14, 529.76, 176) mm, rotated rx 180 ry 0 rz 160 deg; joints [9.479, 55.784, -7.971, -142.659, 54.224, 155.962]
  Set speed (17.6 mm/s)
  Call Extruder(1029.35723)
  MoveL 9797 to (520.96, 530.6, 176) mm, rotated rx 180 ry 0 rz 160 deg; joints [9.602, 55.593, -7.613, -142.593, 54.407, 156.006]
  Set speed (17.6 mm/s)
  Call Extruder(1031.74790)
  MoveL 9798 to (520.34, 531.01, 176) mm, rotated rx 180 ry 0 rz 160 deg; joints [9.664, 55.493, -7.425, -142.562, 54.502, 156.032]
  Set speed (17.6 mm/s)
  Call Extruder(1034.24681)
  MoveL 9799 to (519.69, 531.43, 176) mm, rotated rx 180 ry 0 rz 160 deg; joints [9.727, 55.386, -7.225, -142.532, 54.602, 156.061]
  Set speed (17.6 mm/s)
  Call Extruder(1036.67539)
  MoveL 9800 to (519.04, 531.83, 176) mm, rotated rx -180 ry 0 rz 160 deg; joints [9.787, 55.281, -7.028, -142.505, 54.699, 156.09]
  Set speed (17.6 mm/s)
  Call Extruder(1041.49855)
  MoveL 9801 to (517.74, 532.57, 176) mm, rotated rx 180 ry 0 rz 160 deg; joints [9.903, 55.068, -6.628, -142.456, 54.894, 156.155]
  Set speed (17.6 mm/s)
  Call Extruder(1043.98352)
  MoveL 9802 to (517.05, 532.94, 176) mm, rotated rx 180 ry 0 rz 160 deg; joints [9.96, 54.956, -6.417, -142.433, 54.995, 156.191]
  Call Extruder(1046.60987)
  MoveL 9803 to (516.32, 533.31, 176) mm, rotated rx 180 ry 0 rz 160 deg; joints [10.02, 54.836, -6.192, -142.412, 55.103, 156.231]
  Set speed (17.6 mm/s)
  Call Extruder(1049.12714)
  MoveL 9804 to (515.61, 533.64, 176) mm, rotated rx 180 ry 0 rz 160 deg; joints [10.075, 54.719, -5.974, -142.393, 55.206, 156.272]
  Call Extruder(1053.94681)
  MoveL 9805 to (514.24, 534.25, 176) mm, rotated rx 180 ry 0 rz 160 deg; joints [10.176, 54.493, -5.549, -142.364, 55.404, 156.355]
  Set speed (17.6 mm/s)
  Call Extruder(1058.81476)
  MoveL 9806 to (512.83, 534.8, 176) mm, rotated rx 180 ry 0 rz 160 deg; joints [10.273, 54.259, -5.11, -142.342, 55.604, 156.446]
  Call Extruder(1063.71140)
  MoveL 9807 to (511.38, 535.3, 176) mm, rotated rx -180 ry 0 rz 160 deg; joints [10.365, 54.019, -4.662, -142.328, 55.806, 156.543]
  Set speed (17.6 mm/s)
  Call Extruder(1068.55554)
  MoveL 9808 to (509.94, 535.73, 176) mm, rotated rx 180 ry 0 rz 160 deg; joints [10.449, 53.779, -4.21, -142.322, 56.007, 156.646]
  Set speed (17.6 mm/s)
  Call Extruder(1070.62659)
  MoveL 9809 to (509.32, 535.9, 176) mm, rotated rx -180 ry 0 rz 160 deg; joints [10.483, 53.675, -4.016, -142.322, 56.092, 156.692]
  Set speed (17.6 mm/s)
  Call Extruder(1073.54751)
  MoveL 9810 to (508.43, 536.12, 176) mm, rotated rx 180 ry 0 rz 160 deg; joints [10.529, 53.528, -3.74, -142.323, 56.212, 156.758]
  Set speed (17.6 mm/s)
  Call Extruder(1078.43017)
  MoveL 9811 to (506.95, 536.43, 176) mm, rotated rx 180 ry 0 rz 160 deg; joints [10.601, 53.279, -3.274, -142.332, 56.412, 156.874]
  Set speed (17.6 mm/s)
  Call Extruder(1083.37174)
  MoveL 9812 to (505.43, 536.69, 176) mm, rotated rx -180 ry 0 rz 160 deg; joints [10.667, 53.024, -2.797, -142.35, 56.614, 156.997]
  Set speed (17.6 mm/s)
  Call Extruder(1088.15195)
  MoveL 9813 to (503.95, 536.88, 176) mm, rotated rx 180 ry 0 rz 160 deg; joints [10.724, 52.776, -2.332, -142.373, 56.808, 157.12]
  Set speed (17.6 mm/s)
  Call Extruder(1093.06382)
  MoveL 9814 to (502.43, 537.01, 176) mm, rotated rx -180 ry 0 rz 160 deg; joints [10.775, 52.519, -1.851, -142.406, 57.006, 157.253]
  Set speed (17.6 mm/s)
  Call Extruder(1097.98722)
  MoveL 9815 to (500.89, 537.08, 176) mm, rotated rx 180 ry 0 rz 160 deg; joints [10.82, 52.26, -1.366, -142.447, 57.202, 157.391]
  Set speed (17.6 mm/s)
  Call Extruder(1102.67893)
  MoveL 9816 to (499.43, 537.08, 176) mm, rotated rx 180 ry 0 rz 160 deg; joints [10.855, 52.012, -0.902, -142.492, 57.387, 157.526]
  Set speed (10.0 mm/s)
  MoveL 9817 to (499.43, 537.08, 180) mm, rotated rx 180 ry 0 rz 160 deg; joints [10.855, 51.476, -0.837, -142.307, 57.013, 157.184]
  Set speed (120.0 mm/s)
  MoveL 9818 to (499.42, 536.28, 180) mm, rotated rx -180 ry 0 rz 160 deg; joints [10.756, 51.448, -0.785, -142.425, 56.994, 157.261]
  Set speed (17.7 mm/s)
  Call Extruder(1107.46084)
  MoveL 9819 to (497.92, 536.23, 180) mm, rotated rx 180 ry 0 rz 160 deg; joints [10.784, 51.192, -0.308, -142.481, 57.18, 157.404]
  Set speed (17.7 mm/s)
  Call Extruder(1112.22592)
  MoveL 9820 to (496.43, 536.11, 180) mm, rotated rx -180 ry 0 rz 160 deg; joints [10.805, 50.936, 0.166, -142.544, 57.362, 157.55]
  Set speed (17.7 mm/s)
  Call Extruder(1116.88874)
  MoveL 9821 to (494.98, 535.94, 180) mm, rotated rx -180 ry 0 rz 160 deg; joints [10.818, 50.687, 0.63, -142.612, 57.537, 157.697]
  Set speed (17.7 mm/s)
  Call Extruder(1121.45171)
  MoveL 9822 to (493.56, 535.71, 180) mm, rotated rx 180 ry 0 rz 160 deg; joints [10.824, 50.443, 1.082, -142.687, 57.705, 157.844]
  Call Extruder(1126.45407)
  MoveL 9823 to (492.02, 535.4, 180) mm, rotated rx 180 ry 0 rz 160 deg; joints [10.822, 50.178, 1.576, -142.776, 57.885, 158.008]
  Set speed (17.7 mm/s)
  Call Extruder(1131.06926)
  MoveL 9824 to (490.62, 535.05, 180) mm, rotated rx 180 ry 0 rz 160 deg; joints [10.812, 49.934, 2.028, -142.866, 58.048, 158.162]
  Set speed (17.7 mm/s)
  Call Extruder(1135.80555)
  MoveL 9825 to (489.19, 534.64, 180) mm, rotated rx -180 ry 0 rz 160 deg; joints [10.794, 49.686, 2.489, -142.965, 58.211, 158.323]
  Set speed (17.7 mm/s)
  Call Extruder(1140.59867)
  MoveL 9826 to (487.77, 534.16, 180) mm, rotated rx 180 ry 0 rz 160 deg; joints [10.768, 49.437, 2.951, -143.072, 58.371, 158.489]
  Set speed (17.7 mm/s)
  Call Extruder(1145.15364)
  MoveL 9827 to (486.43, 533.66, 180) mm, rotated rx 180 ry 0 rz 160 deg; joints [10.736, 49.203, 3.385, -143.181, 58.52, 158.648]
  Set speed (17.7 mm/s)
  Call Extruder(1150.07215)
  MoveL 9828 to (485.02, 533.05, 180) mm, rotated rx -180 ry 0 rz 160 deg; joints [10.693, 48.954, 3.847, -143.306, 58.675, 158.822]
  Set speed (17.7 mm/s)
  Call Extruder(1153.31841)
  MoveL 9829 to (484.09, 532.62, 180) mm, rotated rx 180 ry 0 rz 160 deg; joints [10.66, 48.791, 4.149, -143.392, 58.775, 158.938]
  Set speed (17.7 mm/s)
  Call Extruder(1157.10131)
  MoveL 9830 to (483.04, 532.08, 180) mm, rotated rx 180 ry 0 rz 160 deg; joints [10.616, 48.603, 4.497, -143.498, 58.888, 159.074]
  Set speed (17.7 mm/s)
  Call Extruder(1159.51433)
  MoveL 9831 to (482.37, 531.72, 180) mm, rotated rx -180 ry 0 rz 160 deg; joints [10.586, 48.485, 4.716, -143.567, 58.958, 159.161]
  Set speed (17.7 mm/s)
  Call Extruder(1162.08432)
  MoveL 9832 to (481.67, 531.32, 180) mm, rotated rx 180 ry 0 rz 160 deg; joints [10.552, 48.36, 4.947, -143.643, 59.031, 159.254]
  Set speed (17.7 mm/s)
  Call Extruder(1166.40669)
  MoveL 9833 to (480.51, 530.61, 180) mm, rotated rx 180 ry 0 rz 160 deg; joints [10.488, 48.154, 5.33, -143.774, 59.151, 159.411]
  Set speed (17.7 mm/s)
  Call Extruder(1168.92173)
  MoveL 9834 to (479.85, 530.18, 180) mm, rotated rx -180 ry 0 rz 160 deg; joints [10.448, 48.035, 5.549, -143.853, 59.219, 159.503]
  Set speed (17.7 mm/s)
  Call Extruder(1171.35980)
  MoveL 9835 to (479.22, 529.75, 180) mm, rotated rx 180 ry 0 rz 160 deg; joints [10.408, 47.921, 5.76, -143.931, 59.283, 159.592]
  Call Extruder(1173.92549)
  MoveL 9836 to (478.57, 529.28, 180) mm, rotated rx 180 ry 0 rz 160 deg; joints [10.363, 47.803, 5.979, -144.016, 59.348, 159.686]
  Set speed (17.7 mm/s)
  Call Extruder(1178.43629)
  MoveL 9837 to (477.44, 528.42, 180) mm, rotated rx 180 ry 0 rz 160 deg; joints [10.278, 47.599, 6.357, -144.168, 59.46, 159.851]
  Set speed (17.7 mm/s)
  Call Extruder(1183.05790)
  MoveL 9838 to (476.32, 527.5, 180) mm, rotated rx 180 ry 0 rz 160 deg; joints [10.184, 47.396, 6.733, -144.33, 59.568, 160.021]
  Call Extruder(1185.53869)
  MoveL 9839 to (475.74, 526.98, 180) mm, rotated rx 180 ry 0 rz 160 deg; joints [10.131, 47.289, 6.931, -144.42, 59.624, 160.112]
  Call Extruder(1187.89235)
  MoveL 9840 to (475.19, 526.48, 180) mm, rotated rx -180 ry 0 rz 160 deg; joints [10.078, 47.189, 7.116, -144.506, 59.675, 160.198]
  Set speed (17.7 mm/s)
  Call Extruder(1190.24523)
  MoveL 9841 to (474.66, 525.97, 180) mm, rotated rx -180 ry 0 rz 160 deg; joints [10.023, 47.09, 7.298, -144.594, 59.725, 160.284]
  Set speed (17.7 mm/s)
  Call Extruder(1194.79540)
  MoveL 9842 to (473.66, 524.96, 180) mm, rotated rx 180 ry 0 rz 160 deg; joints [9.913, 46.904, 7.642, -144.767, 59.817, 160.45]
  Set speed (17.7 mm/s)
  Call Extruder(1198.10421)
  MoveL 9843 to (472.96, 524.2, 180) mm, rotated rx 180 ry 0 rz 160 deg; joints [9.829, 46.773, 7.885, -144.896, 59.88, 160.57]
  Set speed (17.7 mm/s)
  Call Extruder(1201.59993)
  MoveL 9844 to (472.24, 523.37, 180) mm, rotated rx -180 ry 0 rz 160 deg; joints [9.737, 46.638, 8.134, -145.035, 59.943, 160.697]
  Call Extruder(1205.13312)
  MoveL 9845 to (471.54, 522.51, 180) mm, rotated rx -180 ry 0 rz 160 deg; joints [9.639, 46.506, 8.379, -145.179, 60.002, 160.824]
  Set speed (17.7 mm/s)
  Call Extruder(1209.17947)
  MoveL 9846 to (470.77, 521.5, 180) mm, rotated rx -180 ry 0 rz 160 deg; joints [9.522, 46.359, 8.65, -145.346, 60.067, 160.97]
  Set speed (17.7 mm/s)
  Call Extruder(1211.59516)
  MoveL 9847 to (470.33, 520.89, 180) mm, rotated rx 180 ry 0 rz 160 deg; joints [9.45, 46.274, 8.807, -145.448, 60.103, 161.056]
  Call Extruder(1213.95744)
  MoveL 9848 to (469.91, 520.28, 180) mm, rotated rx -180 ry 0 rz 160 deg; joints [9.379, 46.193, 8.957, -145.549, 60.136, 161.14]
  Set speed (17.7 mm/s)
  Call Extruder(1216.32167)
  MoveL 9849 to (469.5, 519.66, 180) mm, rotated rx 180 ry 0 rz 160 deg; joints [9.305, 46.114, 9.104, -145.651, 60.168, 161.224]
  Set speed (17.7 mm/s)
  Call Extruder(1218.69385)
  MoveL 9850 to (469.11, 519.03, 180) mm, rotated rx 180 ry 0 rz 160 deg; joints [9.23, 46.036, 9.247, -145.755, 60.198, 161.307]
  Set speed (17.7 mm/s)
  Call Extruder(1222.79786)
  MoveL 9851 to (468.45, 517.92, 180) mm, rotated rx -180 ry 0 rz 160 deg; joints [9.096, 45.907, 9.486, -145.936, 60.246, 161.45]
  Set speed (17.7 mm/s)
  Call Extruder(1228.10128)
  MoveL 9852 to (467.66, 516.46, 180) mm, rotated rx -180 ry 0 rz 160 deg; joints [8.917, 45.748, 9.778, -146.174, 60.3, 161.634]
  Set speed (17.7 mm/s)
  Call Extruder(1231.62112)
  MoveL 9853 to (467.18, 515.47, 180) mm, rotated rx -180 ry 0 rz 160 deg; joints [8.794, 45.65, 9.96, -146.335, 60.331, 161.753]
  Set speed (17.7 mm/s)
  Call Extruder(1235.09827)
  MoveL 9854 to (466.73, 514.48, 180) mm, rotated rx 180 ry 0 rz 160 deg; joints [8.67, 45.557, 10.132, -146.495, 60.358, 161.871]
  Set speed (17.7 mm/s)
  Call Extruder(1239.92183)
  MoveL 9855 to (466.15, 513.08, 180) mm, rotated rx 180 ry 0 rz 160 deg; joints [8.493, 45.435, 10.356, -146.721, 60.389, 162.031]
  Set speed (17.7 mm/s)
  Call Extruder(1244.61472)
  MoveL 9856 to (465.65, 511.7, 180) mm, rotated rx 180 ry 0 rz 160 deg; joints [8.316, 45.326, 10.557, -146.943, 60.411, 162.185]
  Set speed (17.7 mm/s)
  Call Extruder(1249.49920)
  MoveL 9857 to (465.19, 510.24, 180) mm, rotated rx -180 ry 0 rz 160 deg; joints [8.128, 45.222, 10.749, -147.176, 60.428, 162.342]
  Set speed (17.7 mm/s)
  Call Extruder(1254.20490)
  MoveL 9858 to (464.8, 508.81, 180) mm, rotated rx -180 ry 0 rz 160 deg; joints [7.942, 45.131, 10.916, -147.403, 60.436, 162.49]
  Set speed (17.7 mm/s)
  Call Extruder(1258.82509)
  MoveL 9859 to (464.48, 507.4, 180) mm, rotated rx 180 ry 0 rz 160 deg; joints [7.756, 45.052, 11.062, -147.628, 60.437, 162.631]
  Set speed (17.7 mm/s)
  Call Extruder(1263.70049)
  MoveL 9860 to (464.2, 505.9, 180) mm, rotated rx 180 ry 0 rz 160 deg; joints [7.557, 44.978, 11.199, -147.866, 60.431, 162.778]
  Call Extruder(1268.43813)
  MoveL 9861 to (463.98, 504.43, 180) mm, rotated rx 180 ry 0 rz 160 deg; joints [7.36, 44.916, 11.314, -148.097, 60.417, 162.917]
  Set speed (17.7 mm/s)
  Call Extruder(1273.17222)
  MoveL 9862 to (463.84, 502.95, 180) mm, rotated rx -180 ry 0 rz 160 deg; joints [7.161, 44.864, 11.409, -148.329, 60.396, 163.051]
  Set speed (17.7 mm/s)
  Call Extruder(1277.72950)
  MoveL 9863 to (463.75, 501.52, 180) mm, rotated rx 180 ry 0 rz 160 deg; joints [6.968, 44.823, 11.484, -148.552, 60.369, 163.177]
  Set speed (17.7 mm/s)
  Call Extruder(1282.56309)
  MoveL 9864 to (463.72, 500.01, 180) mm, rotated rx 180 ry 0 rz 160 deg; joints [6.761, 44.79, 11.545, -148.788, 60.333, 163.306]
  Call Extruder(1286.90226)
  MoveL 9865 to (463.74, 498.65, 180) mm, rotated rx 180 ry 0 rz 160 deg; joints [6.575, 44.77, 11.583, -148.999, 60.294, 163.419]
  Set speed (17.7 mm/s)
  Call Extruder(1290.98729)
  MoveL 9866 to (463.81, 497.37, 180) mm, rotated rx -180 ry 0 rz 160 deg; joints [6.398, 44.758, 11.604, -149.197, 60.253, 163.521]
  Set speed (17.7 mm/s)
  Call Extruder(1295.32214)
  MoveL 9867 to (463.93, 496.01, 180) mm, rotated rx 180 ry 0 rz 160 deg; joints [6.211, 44.754, 11.612, -149.405, 60.203, 163.626]
  Set speed (17.7 mm/s)
  Call Extruder(1299.57947)
  MoveL 9868 to (464.1, 494.69, 180) mm, rotated rx 180 ry 0 rz 160 deg; joints [6.027, 44.759, 11.603, -149.607, 60.148, 163.725]
  Call Extruder(1303.91519)
  MoveL 9869 to (464.33, 493.35, 180) mm, rotated rx 180 ry 0 rz 160 deg; joints [5.84, 44.772, 11.579, -149.811, 60.086, 163.821]
  Set speed (17.7 mm/s)
  Call Extruder(1308.03723)
  MoveL 9870 to (464.59, 492.08, 180) mm, rotated rx 180 ry 0 rz 160 deg; joints [5.663, 44.792, 11.541, -150.002, 60.022, 163.909]
  Set speed (17.7 mm/s)
  Call Extruder(1312.36171)
  MoveL 9871 to (464.91, 490.76, 180) mm, rotated rx 180 ry 0 rz 160 deg; joints [5.478, 44.821, 11.487, -150.201, 59.949, 163.998]
  Set speed (17.7 mm/s)
  Call Extruder(1316.53108)
  MoveL 9872 to (465.27, 489.51, 180) mm, rotated rx 180 ry 0 rz 160 deg; joints [5.301, 44.858, 11.42, -150.388, 59.873, 164.079]
  Set speed (17.7 mm/s)
  Call Extruder(1320.73005)
  MoveL 9873 to (465.67, 488.25, 180) mm, rotated rx 180 ry 0 rz 160 deg; joints [5.124, 44.903, 11.338, -150.574, 59.792, 164.156]
  Set speed (17.7 mm/s)
  Call Extruder(1325.17702)
  MoveL 9874 to (466.15, 486.94, 180) mm, rotated rx 180 ry 0 rz 160 deg; joints [4.939, 44.958, 11.235, -150.767, 59.701, 164.233]
  Set speed (17.7 mm/s)
  Call Extruder(1328.58484)
  MoveL 9875 to (466.54, 485.95, 180) mm, rotated rx 180 ry 0 rz 160 deg; joints [4.799, 45.007, 11.146, -150.912, 59.627, 164.289]
  Call Extruder(1333.70004)
  MoveL 9876 to (467.2, 484.49, 180) mm, rotated rx 180 ry 0 rz 160 deg; joints [4.591, 45.09, 10.993, -151.124, 59.51, 164.367]
  Set speed (17.7 mm/s)
  Call Extruder(1337.96659)
  MoveL 9877 to (467.79, 483.29, 180) mm, rotated rx 180 ry 0 rz 160 deg; joints [4.421, 45.167, 10.851, -151.296, 59.407, 164.428]
  Set speed (17.7 mm/s)
  Call Extruder(1342.11861)
  MoveL 9878 to (468.41, 482.15, 180) mm, rotated rx 180 ry 0 rz 160 deg; joints [4.258, 45.249, 10.698, -151.458, 59.303, 164.482]
  Set speed (17.7 mm/s)
  Call Extruder(1346.26951)
  MoveL 9879 to (469.07, 481.02, 180) mm, rotated rx -180 ry 0 rz 160 deg; joints [4.099, 45.339, 10.533, -151.615, 59.193, 164.531]
  Set speed (17.7 mm/s)
  Call Extruder(1350.65019)
  MoveL 9880 to (469.81, 479.87, 180) mm, rotated rx 180 ry 0 rz 160 deg; joints [3.934, 45.442, 10.343, -151.775, 59.073, 164.578]
  Call Extruder(1354.96795)
  MoveL 9881 to (470.58, 478.75, 180) mm, rotated rx -180 ry 0 rz 160 deg; joints [3.776, 45.55, 10.144, -151.928, 58.95, 164.619]
  Call Extruder(1359.30481)
  MoveL 9882 to (471.4, 477.67, 180) mm, rotated rx 180 ry 0 rz 160 deg; joints [3.621, 45.667, 9.928, -152.074, 58.822, 164.655]
  Call Extruder(1363.42340)
  MoveL 9883 to (472.22, 476.66, 180) mm, rotated rx -180 ry 0 rz 160 deg; joints [3.478, 45.785, 9.711, -152.207, 58.696, 164.684]
  Call Extruder(1367.62015)
  MoveL 9884 to (473.08, 475.67, 180) mm, rotated rx 180 ry 0 rz 160 deg; joints [3.337, 45.911, 9.478, -152.336, 58.565, 164.709]
  Set speed (17.7 mm/s)
  Call Extruder(1372.08734)
  MoveL 9885 to (474.04, 474.65, 180) mm, rotated rx -180 ry 0 rz 160 deg; joints [3.192, 46.052, 9.217, -152.467, 58.42, 164.73]
  Set speed (17.7 mm/s)
  Call Extruder(1376.29806)
  MoveL 9886 to (474.98, 473.72, 180) mm, rotated rx -180 ry 0 rz 160 deg; joints [3.06, 46.192, 8.958, -152.582, 58.28, 164.745]
  Call Extruder(1380.39545)
  MoveL 9887 to (475.93, 472.85, 180) mm, rotated rx -180 ry 0 rz 160 deg; joints [2.936, 46.335, 8.695, -152.688, 58.141, 164.753]
  Set speed (17.7 mm/s)
  Call Extruder(1384.85633)
  MoveL 9888 to (476.99, 471.94, 180) mm, rotated rx -180 ry 0 rz 160 deg; joints [2.807, 46.495, 8.398, -152.796, 57.985, 164.757]
  Set speed (17.7 mm/s)
  Call Extruder(1389.03566)
  MoveL 9889 to (478.02, 471.13, 180) mm, rotated rx 180 ry 0 rz 160 deg; joints [2.692, 46.652, 8.108, -152.89, 57.837, 164.755]
  Set speed (17.7 mm/s)
  Call Extruder(1393.40127)
  MoveL 9890 to (479.12, 470.32, 180) mm, rotated rx 180 ry 0 rz 160 deg; joints [2.577, 46.822, 7.794, -152.979, 57.678, 164.748]
  Set speed (17.7 mm/s)
  Call Extruder(1397.55128)
  MoveL 9891 to (480.2, 469.59, 180) mm, rotated rx -180 ry 0 rz 160 deg; joints [2.473, 46.989, 7.486, -153.057, 57.525, 164.735]
  Set speed (17.7 mm/s)
  Call Extruder(1401.75335)
  MoveL 9892 to (481.32, 468.89, 180) mm, rotated rx -180 ry 0 rz 160 deg; joints [2.374, 47.163, 7.164, -153.128, 57.367, 164.717]
  Set speed (17.7 mm/s)
  Call Extruder(1405.90389)
  MoveL 9893 to (482.44, 468.24, 180) mm, rotated rx 180 ry 0 rz 160 deg; joints [2.281, 47.339, 6.837, -153.19, 57.208, 164.694]
  Set speed (17.7 mm/s)
  Call Extruder(1411.27723)
  MoveL 9894 to (483.93, 467.46, 180) mm, rotated rx 180 ry 0 rz 160 deg; joints [2.17, 47.575, 6.402, -153.26, 57.001, 164.656]
  Call Extruder(1414.51814)
  MoveL 9895 to (484.85, 467.03, 180) mm, rotated rx 180 ry 0 rz 160 deg; joints [2.109, 47.72, 6.132, -153.294, 56.873, 164.628]
  Set speed (17.7 mm/s)
  Call Extruder(1418.96400)
  MoveL 9896 to (486.13, 466.47, 180) mm, rotated rx 180 ry 0 rz 160 deg; joints [2.029, 47.924, 5.755, -153.335, 56.697, 164.585]
  Call Extruder(1423.12691)
  MoveL 9897 to (487.35, 465.99, 180) mm, rotated rx 180 ry 0 rz 160 deg; joints [1.961, 48.119, 5.395, -153.365, 56.531, 164.539]
  Set speed (17.7 mm/s)
  Call Extruder(1427.44563)
  MoveL 9898 to (488.62, 465.54, 180) mm, rotated rx -180 ry 0 rz 160 deg; joints [1.897, 48.325, 5.013, -153.387, 56.357, 164.486]
  Set speed (17.7 mm/s)
  Call Extruder(1431.68599)
  MoveL 9899 to (489.89, 465.15, 180) mm, rotated rx 180 ry 0 rz 160 deg; joints [1.84, 48.53, 4.632, -153.4, 56.185, 164.428]
  Set speed (17.7 mm/s)
  Call Extruder(1435.89738)
  MoveL 9900 to (491.17, 464.81, 180) mm, rotated rx -180 ry 0 rz 160 deg; joints [1.79, 48.738, 4.247, -153.405, 56.013, 164.364]
  Call Extruder(1440.24647)
  MoveL 9901 to (492.5, 464.5, 180) mm, rotated rx 180 ry 0 rz 160 deg; joints [1.745, 48.956, 3.843, -153.401, 55.834, 164.293]
  Set speed (17.7 mm/s)
  Call Extruder(1444.36352)
  MoveL 9902 to (493.77, 464.26, 180) mm, rotated rx -180 ry 0 rz 160 deg; joints [1.708, 49.164, 3.456, -153.389, 55.665, 164.221]
  Set speed (17.7 mm/s)
  Call Extruder(1448.32998)
  MoveL 9903 to (494.99, 464.06, 180) mm, rotated rx 180 ry 0 rz 160 deg; joints [1.678, 49.367, 3.08, -153.371, 55.502, 164.146]
  Call Extruder(1452.99335)
  MoveL 9904 to (496.45, 463.89, 180) mm, rotated rx -180 ry 0 rz 160 deg; joints [1.651, 49.609, 2.632, -153.339, 55.309, 164.052]
  Set speed (17.7 mm/s)
  Call Extruder(1457.21240)
  MoveL 9905 to (497.76, 463.78, 180) mm, rotated rx 180 ry 0 rz 160 deg; joints [1.632, 49.829, 2.223, -153.302, 55.136, 163.961]
  Call Extruder(1461.53648)
  MoveL 9906 to (499.12, 463.73, 180) mm, rotated rx 180 ry 0 rz 160 deg; joints [1.62, 50.057, 1.8, -153.255, 54.958, 163.862]
  Set speed (17.7 mm/s)
  Call Extruder(1465.73402)
  MoveL 9907 to (500.44, 463.72, 180) mm, rotated rx 180 ry 0 rz 160 deg; joints [1.614, 50.279, 1.387, -153.201, 54.786, 163.761]
  Set speed (17.7 mm/s)
  Call Extruder(1470.07188)
  MoveL 9908 to (501.8, 463.76, 180) mm, rotated rx -180 ry 0 rz 160 deg; joints [1.615, 50.51, 0.958, -153.137, 54.61, 163.651]
  Set speed (17.7 mm/s)
  Call Extruder(1474.25561)
  MoveL 9909 to (503.11, 463.85, 180) mm, rotated rx 180 ry 0 rz 160 deg; joints [1.621, 50.734, 0.543, -153.068, 54.44, 163.54]
  Set speed (17.7 mm/s)
  Call Extruder(1478.57218)
  MoveL 9910 to (504.45, 463.99, 180) mm, rotated rx -180 ry 0 rz 160 deg; joints [1.634, 50.965, 0.113, -152.988, 54.267, 163.421]
  Set speed (17.7 mm/s)
  Call Extruder(1482.67975)
  MoveL 9911 to (505.73, 464.17, 180) mm, rotated rx -180 ry 0 rz 160 deg; joints [1.653, 51.185, -0.295, -152.904, 54.104, 163.302]
  Set speed (17.7 mm/s)
  Call Extruder(1487.04671)
  MoveL 9912 to (507.08, 464.41, 180) mm, rotated rx -180 ry 0 rz 160 deg; joints [1.678, 51.418, -0.73, -152.808, 53.933, 163.171]
  Set speed (17.7 mm/s)
  Call Extruder(1490.68921)
  MoveL 9913 to (508.19, 464.65, 180) mm, rotated rx 180 ry 0 rz 160 deg; joints [1.704, 51.613, -1.092, -152.721, 53.792, 163.058]
  Set speed (17.7 mm/s)
  Call Extruder(1495.53219)
  MoveL 9914 to (509.66, 465.03, 180) mm, rotated rx 180 ry 0 rz 160 deg; joints [1.745, 51.871, -1.572, -152.597, 53.606, 162.903]
  Set speed (17.7 mm/s)
  Call Extruder(1499.81137)
  MoveL 9915 to (510.95, 465.41, 180) mm, rotated rx 180 ry 0 rz 160 deg; joints [1.788, 52.098, -1.995, -152.48, 53.445, 162.761]
  Set speed (17.7 mm/s)
  Call Extruder(1504.12928)
  MoveL 9916 to (512.24, 465.84, 180) mm, rotated rx 180 ry 0 rz 160 deg; joints [1.837, 52.326, -2.419, -152.354, 53.286, 162.612]
  Set speed (17.7 mm/s)
  Call Extruder(1508.31202)
  MoveL 9917 to (513.46, 466.31, 180) mm, rotated rx 180 ry 0 rz 160 deg; joints [1.889, 52.546, -2.828, -152.226, 53.134, 162.465]
  Set speed (17.7 mm/s)
  Call Extruder(1512.65564)
  MoveL 9918 to (514.72, 466.83, 180) mm, rotated rx -180 ry 0 rz 160 deg; joints [1.949, 52.771, -3.248, -152.086, 52.981, 162.308]
  Set speed (17.7 mm/s)
  Call Extruder(1516.66636)
  MoveL 9919 to (515.86, 467.36, 180) mm, rotated rx -180 ry 0 rz 160 deg; joints [2.01, 52.978, -3.632, -151.951, 52.842, 162.16]
  Call Extruder(1521.08189)
  MoveL 9920 to (517.09, 467.99, 180) mm, rotated rx -180 ry 0 rz 160 deg; joints [2.081, 53.202, -4.051, -151.795, 52.693, 161.994]
  Set speed (17.7 mm/s)
  Call Extruder(1525.42290)
  MoveL 9921 to (518.28, 468.66, 180) mm, rotated rx -180 ry 0 rz 160 deg; joints [2.157, 53.42, -4.457, -151.636, 52.551, 161.826]
  Set speed (17.7 mm/s)
  Call Extruder(1529.58990)
  MoveL 9922 to (519.4, 469.34, 180) mm, rotated rx -180 ry 0 rz 160 deg; joints [2.235, 53.626, -4.841, -151.478, 52.419, 161.663]
  Set speed (17.7 mm/s)
  Call Extruder(1533.80114)
  MoveL 9923 to (520.5, 470.06, 180) mm, rotated rx 180 ry 0 rz 160 deg; joints [2.318, 53.832, -5.224, -151.313, 52.289, 161.494]
  Set speed (17.7 mm/s)
  Call Extruder(1538.13185)
  MoveL 9924 to (521.61, 470.85, 180) mm, rotated rx 180 ry 0 rz 160 deg; joints [2.409, 54.039, -5.61, -151.138, 52.161, 161.319]
  Set speed (17.7 mm/s)
  Call Extruder(1542.41940)
  MoveL 9925 to (522.67, 471.67, 180) mm, rotated rx -180 ry 0 rz 160 deg; joints [2.502, 54.24, -5.986, -150.96, 52.039, 161.143]
  Set speed (17.7 mm/s)
  Call Extruder(1546.63276)
  MoveL 9926 to (523.69, 472.51, 180) mm, rotated rx -180 ry 0 rz 160 deg; joints [2.599, 54.434, -6.347, -150.78, 51.924, 160.968]
  Set speed (17.7 mm/s)
  Call Extruder(1550.99012)
  MoveL 9927 to (524.71, 473.43, 180) mm, rotated rx -180 ry 0 rz 160 deg; joints [2.704, 54.629, -6.711, -150.589, 51.811, 160.785]
  Set speed (17.7 mm/s)
  Call Extruder(1555.31405)
  MoveL 9928 to (525.69, 474.37, 180) mm, rotated rx -180 ry 0 rz 160 deg; joints [2.811, 54.819, -7.065, -150.396, 51.703, 160.602]
  Call Extruder(1560.27150)
  MoveL 9929 to (526.76, 475.49, 180) mm, rotated rx 180 ry 0 rz 160 deg; joints [2.94, 55.029, -7.458, -150.17, 51.588, 160.391]
  Set speed (17.7 mm/s)
  Call Extruder(1564.55634)
  MoveL 9930 to (527.65, 476.5, 180) mm, rotated rx -180 ry 0 rz 160 deg; joints [3.055, 55.205, -7.786, -149.971, 51.495, 160.207]
  Set speed (17.7 mm/s)
  Call Extruder(1567.01056)
  MoveL 9931 to (528.14, 477.09, 180) mm, rotated rx 180 ry 0 rz 160 deg; joints [3.123, 55.303, -7.969, -149.855, 51.444, 160.102]
  Call Extruder(1569.36736)
  MoveL 9932 to (528.6, 477.67, 180) mm, rotated rx -180 ry 0 rz 160 deg; joints [3.189, 55.396, -8.142, -149.744, 51.398, 160.001]
  Call Extruder(0.00000)
  Call Extruder(4.64330)
  MoveL 9933 to (529.48, 478.84, 180) mm, rotated rx -180 ry 0 rz 160 deg; joints [3.323, 55.573, -8.472, -149.521, 51.311, 159.802]
  Call Extruder(7.08951)
  MoveL 9934 to (529.92, 479.47, 180) mm, rotated rx 180 ry 0 rz 160 deg; joints [3.394, 55.663, -8.641, -149.403, 51.269, 159.697]
  Set speed (17.7 mm/s)
  Call Extruder(9.47796)
  MoveL 9935 to (530.33, 480.09, 180) mm, rotated rx 180 ry 0 rz 160 deg; joints [3.466, 55.749, -8.802, -149.287, 51.229, 159.594]
  Set speed (17.7 mm/s)
  Call Extruder(11.83361)
  MoveL 9936 to (530.73, 480.71, 180) mm, rotated rx 180 ry 0 rz 160 deg; joints [3.537, 55.832, -8.957, -149.172, 51.192, 159.494]
  Call Extruder(16.57096)
  MoveL 9937 to (531.5, 481.98, 180) mm, rotated rx -180 ry 0 rz 160 deg; joints [3.682, 55.993, -9.256, -148.94, 51.124, 159.292]
  Set speed (17.7 mm/s)
  Call Extruder(20.25652)
  MoveL 9938 to (532.06, 482.99, 180) mm, rotated rx -180 ry 0 rz 160 deg; joints [3.798, 56.112, -9.479, -148.758, 51.076, 159.136]
  Call Extruder(23.82915)
  MoveL 9939 to (532.57, 483.99, 180) mm, rotated rx -180 ry 0 rz 160 deg; joints [3.912, 56.222, -9.685, -148.58, 51.035, 158.986]
  Set speed (17.7 mm/s)
  Call Extruder(27.01691)
  MoveL 9940 to (532.99, 484.89, 180) mm, rotated rx -180 ry 0 rz 160 deg; joints [4.015, 56.316, -9.86, -148.422, 51.003, 158.853]
  Set speed (17.7 mm/s)
  Call Extruder(30.79654)
  MoveL 9941 to (533.46, 485.98, 180) mm, rotated rx -180 ry 0 rz 160 deg; joints [4.139, 56.421, -10.057, -148.234, 50.97, 158.698]
  Set speed (17.7 mm/s)
  Call Extruder(33.03445)
  MoveL 9942 to (533.73, 486.63, 180) mm, rotated rx 180 ry 0 rz 160 deg; joints [4.214, 56.482, -10.171, -148.122, 50.952, 158.606]
  Set speed (17.7 mm/s)
  Call Extruder(37.94288)
  MoveL 9943 to (534.27, 488.07, 180) mm, rotated rx 180 ry 0 rz 160 deg; joints [4.379, 56.607, -10.404, -147.878, 50.921, 158.407]
  Set speed (17.7 mm/s)
  Call Extruder(42.55383)
  MoveL 9944 to (534.72, 489.45, 180) mm, rotated rx 180 ry 0 rz 160 deg; joints [4.537, 56.714, -10.603, -147.648, 50.901, 158.224]
  Set speed (17.7 mm/s)
  Call Extruder(47.21903)
  MoveL 9945 to (535.11, 490.86, 180) mm, rotated rx 180 ry 0 rz 160 deg; joints [4.699, 56.813, -10.788, -147.417, 50.888, 158.042]
  Set speed (17.7 mm/s)
  Call Extruder(51.96034)
  MoveL 9946 to (535.46, 492.3, 180) mm, rotated rx 180 ry 0 rz 160 deg; joints [4.865, 56.904, -10.958, -147.184, 50.884, 157.862]
  Set speed (17.7 mm/s)
  Call Extruder(56.77548)
  MoveL 9947 to (535.75, 493.78, 180) mm, rotated rx -180 ry 0 rz 160 deg; joints [5.036, 56.985, -11.11, -146.949, 50.89, 157.684]
  Set speed (17.7 mm/s)
  Call Extruder(61.49631)
  MoveL 9948 to (535.97, 495.25, 180) mm, rotated rx -180 ry 0 rz 160 deg; joints [5.205, 57.054, -11.239, -146.721, 50.904, 157.515]
  Set speed (17.7 mm/s)
  Call Extruder(66.33440)
  MoveL 9949 to (536.14, 496.75, 180) mm, rotated rx -180 ry 0 rz 160 deg; joints [5.38, 57.114, -11.351, -146.49, 50.928, 157.347]
  Set speed (17.7 mm/s)
  Call Extruder(70.97670)
  MoveL 9950 to (536.24, 498.21, 180) mm, rotated rx -180 ry 0 rz 160 deg; joints [5.548, 57.161, -11.439, -146.271, 50.959, 157.191]
  Set speed (17.7 mm/s)
  Call Extruder(75.70756)
  MoveL 9951 to (536.29, 499.69, 180) mm, rotated rx 180 ry 0 rz 160 deg; joints [5.721, 57.198, -11.508, -146.051, 50.999, 157.039]
  Set speed (17.7 mm/s)
  Call Extruder(80.32930)
  MoveL 9952 to (536.27, 501.14, 180) mm, rotated rx 180 ry 0 rz 160 deg; joints [5.891, 57.223, -11.555, -145.841, 51.048, 156.897]
  Set speed (17.7 mm/s)
  Call Extruder(85.15577)
  MoveL 9953 to (536.19, 502.65, 180) mm, rotated rx -180 ry 0 rz 160 deg; joints [6.068, 57.238, -11.584, -145.625, 51.106, 156.756]
  Call Extruder(89.82053)
  MoveL 9954 to (536.05, 504.11, 180) mm, rotated rx -180 ry 0 rz 160 deg; joints [6.24, 57.243, -11.592, -145.421, 51.171, 156.626]
  Set speed (17.7 mm/s)
  Call Extruder(94.47856)
  MoveL 9955 to (535.86, 505.56, 180) mm, rotated rx -180 ry 0 rz 160 deg; joints [6.412, 57.236, -11.58, -145.221, 51.244, 156.503]
  Set speed (17.7 mm/s)
  Call Extruder(99.34792)
  MoveL 9956 to (535.59, 507.06, 180) mm, rotated rx -180 ry 0 rz 160 deg; joints [6.59, 57.218, -11.545, -145.018, 51.329, 156.384]
  Set speed (17.7 mm/s)
  Call Extruder(104.13283)
  MoveL 9957 to (535.27, 508.53, 180) mm, rotated rx -180 ry 0 rz 160 deg; joints [6.766, 57.188, -11.491, -144.825, 51.42, 156.274]
  Set speed (17.7 mm/s)
  Call Extruder(109.00451)
  MoveL 9958 to (534.88, 510.01, 180) mm, rotated rx 180 ry 0 rz 160 deg; joints [6.944, 57.147, -11.413, -144.633, 51.521, 156.171]
  Set speed (17.7 mm/s)
  Call Extruder(113.44510)
  MoveL 9959 to (534.47, 511.34, 180) mm, rotated rx -180 ry 0 rz 160 deg; joints [7.105, 57.099, -11.323, -144.464, 51.62, 156.085]
  Set speed (17.7 mm/s)
  Call Extruder(118.11088)
  MoveL 9960 to (533.98, 512.72, 180) mm, rotated rx -180 ry 0 rz 160 deg; joints [7.273, 57.038, -11.21, -144.293, 51.731, 156.003]
  Set speed (17.7 mm/s)
  Call Extruder(122.91991)
  MoveL 9961 to (533.43, 514.12, 180) mm, rotated rx 180 ry 0 rz 160 deg; joints [7.445, 56.965, -11.074, -144.122, 51.853, 155.927]
  Set speed (17.7 mm/s)
  Call Extruder(127.79755)
  MoveL 9962 to (532.81, 515.52, 180) mm, rotated rx -180 ry 0 rz 160 deg; joints [7.618, 56.881, -10.917, -143.955, 51.983, 155.857]
  Set speed (17.7 mm/s)
  Call Extruder(132.52668)
  MoveL 9963 to (532.14, 516.84, 180) mm, rotated rx 180 ry 0 rz 160 deg; joints [7.783, 56.787, -10.741, -143.802, 52.116, 155.801]
  Set speed (17.7 mm/s)
  Call Extruder(134.88283)
  MoveL 9964 to (531.79, 517.49, 180) mm, rotated rx 180 ry 0 rz 160 deg; joints [7.864, 56.737, -10.647, -143.727, 52.185, 155.776]
  Call Extruder(137.46481)
  MoveL 9965 to (531.39, 518.2, 180) mm, rotated rx 180 ry 0 rz 160 deg; joints [7.953, 56.68, -10.54, -143.648, 52.262, 155.75]
  Call Extruder(141.99372)
  MoveL 9966 to (530.66, 519.41, 180) mm, rotated rx -180 ry 0 rz 160 deg; joints [8.108, 56.571, -10.337, -143.513, 52.401, 155.713]
  Call Extruder(146.62039)
  MoveL 9967 to (529.86, 520.62, 180) mm, rotated rx 180 ry 0 rz 160 deg; joints [8.263, 56.451, -10.113, -143.383, 52.548, 155.682]
  Call Extruder(149.50566)
  MoveL 9968 to (529.33, 521.36, 180) mm, rotated rx 180 ry 0 rz 160 deg; joints [8.358, 56.372, -9.965, -143.305, 52.643, 155.667]
  Set speed (17.7 mm/s)
  Call Extruder(151.44726)
  MoveL 9969 to (528.97, 521.85, 180) mm, rotated rx 180 ry 0 rz 160 deg; joints [8.422, 56.316, -9.86, -143.254, 52.708, 155.66]
  Set speed (17.7 mm/s)
  Call Extruder(155.81982)
  MoveL 9970 to (528.12, 522.93, 180) mm, rotated rx -180 ry 0 rz 160 deg; joints [8.563, 56.187, -9.618, -143.143, 52.856, 155.646]
  Set speed (17.7 mm/s)
  Call Extruder(158.54967)
  MoveL 9971 to (527.57, 523.59, 180) mm, rotated rx 180 ry 0 rz 160 deg; joints [8.65, 56.101, -9.459, -143.078, 52.951, 155.642]
  Set speed (17.7 mm/s)
  Call Extruder(160.91752)
  MoveL 9972 to (527.09, 524.15, 180) mm, rotated rx 180 ry 0 rz 160 deg; joints [8.725, 56.025, -9.317, -143.023, 53.035, 155.641]
  Set speed (17.7 mm/s)
  Call Extruder(165.54288)
  MoveL 9973 to (526.1, 525.21, 180) mm, rotated rx -180 ry 0 rz 160 deg; joints [8.867, 55.87, -9.028, -142.921, 53.201, 155.644]
  Call Extruder(167.98603)
  MoveL 9974 to (525.56, 525.75, 180) mm, rotated rx -180 ry 0 rz 160 deg; joints [8.941, 55.785, -8.869, -142.87, 53.29, 155.649]
  Set speed (17.7 mm/s)
  Call Extruder(170.39366)
  MoveL 9975 to (525.02, 526.28, 180) mm, rotated rx -180 ry 0 rz 160 deg; joints [9.013, 55.699, -8.709, -142.821, 53.379, 155.657]
  Set speed (17.7 mm/s)
  Call Extruder(172.77878)
  MoveL 9976 to (524.47, 526.79, 180) mm, rotated rx 180 ry 0 rz 160 deg; joints [9.084, 55.612, -8.546, -142.775, 53.468, 155.666]
  Set speed (17.7 mm/s)
  Call Extruder(175.10867)
  MoveL 9977 to (523.93, 527.28, 180) mm, rotated rx -180 ry 0 rz 160 deg; joints [9.152, 55.525, -8.384, -142.732, 53.557, 155.677]
  Set speed (17.7 mm/s)
  Call Extruder(177.38735)
  MoveL 9978 to (523.39, 527.75, 180) mm, rotated rx 180 ry 0 rz 160 deg; joints [9.217, 55.439, -8.222, -142.691, 53.643, 155.689]
  Call Extruder(179.88086)
  MoveL 9979 to (522.78, 528.24, 180) mm, rotated rx 180 ry 0 rz 160 deg; joints [9.288, 55.342, -8.041, -142.649, 53.739, 155.705]
  Set speed (17.7 mm/s)
  Call Extruder(182.19983)
  MoveL 9980 to (522.21, 528.69, 180) mm, rotated rx 180 ry 0 rz 160 deg; joints [9.352, 55.249, -7.869, -142.612, 53.829, 155.723]
  Set speed (17.7 mm/s)
  Call Extruder(186.75033)
  MoveL 9981 to (521.07, 529.54, 180) mm, rotated rx 180 ry 0 rz 160 deg; joints [9.475, 55.064, -7.523, -142.544, 54.007, 155.762]
  Call Extruder(189.30909)
  MoveL 9982 to (520.41, 530, 180) mm, rotated rx -180 ry 0 rz 160 deg; joints [9.543, 54.957, -7.323, -142.509, 54.109, 155.787]
  Set speed (17.7 mm/s)
  Call Extruder(191.60165)
  MoveL 9983 to (519.81, 530.4, 180) mm, rotated rx 180 ry 0 rz 160 deg; joints [9.602, 54.859, -7.141, -142.48, 54.2, 155.811]
  Set speed (17.7 mm/s)
  Call Extruder(196.83475)
  MoveL 9984 to (518.42, 531.27, 180) mm, rotated rx 180 ry 0 rz 160 deg; joints [9.733, 54.631, -6.715, -142.419, 54.41, 155.873]
  Set speed (17.7 mm/s)
  Call Extruder(200.97292)
  MoveL 9985 to (517.29, 531.91, 180) mm, rotated rx -180 ry 0 rz 160 deg; joints [9.833, 54.446, -6.369, -142.377, 54.578, 155.929]
  Set speed (17.7 mm/s)
  Call Extruder(205.04054)
  MoveL 9986 to (516.15, 532.49, 180) mm, rotated rx -180 ry 0 rz 160 deg; joints [9.926, 54.259, -6.022, -142.342, 54.744, 155.989]
  Set speed (17.7 mm/s)
  Call Extruder(208.12433)
  MoveL 9987 to (515.28, 532.91, 180) mm, rotated rx -180 ry 0 rz 160 deg; joints [9.994, 54.116, -5.753, -142.32, 54.87, 156.038]
  Set speed (17.7 mm/s)
  Call Extruder(212.80317)
  MoveL 9988 to (513.94, 533.5, 180) mm, rotated rx 180 ry 0 rz 160 deg; joints [10.093, 53.893, -5.338, -142.291, 55.062, 156.118]
  Set speed (17.7 mm/s)
  Call Extruder(217.60133)
  MoveL 9989 to (512.54, 534.05, 180) mm, rotated rx -180 ry 0 rz 160 deg; joints [10.189, 53.66, -4.904, -142.27, 55.26, 156.207]
  Set speed (17.7 mm/s)
  Call Extruder(222.29879)
  MoveL 9990 to (511.15, 534.53, 180) mm, rotated rx 180 ry 0 rz 160 deg; joints [10.277, 53.428, -4.472, -142.257, 55.454, 156.301]
  Set speed (17.7 mm/s)
  Call Extruder(227.20115)
  MoveL 9991 to (509.68, 534.97, 180) mm, rotated rx 180 ry 0 rz 160 deg; joints [10.363, 53.182, -4.013, -142.251, 55.657, 156.404]
  Set speed (17.7 mm/s)
  Call Extruder(229.02592)
  MoveL 9992 to (509.12, 535.12, 180) mm, rotated rx 180 ry 0 rz 160 deg; joints [10.393, 53.089, -3.84, -142.251, 55.732, 156.445]
  Set speed (17.7 mm/s)
  Call Extruder(231.77129)
  MoveL 9993 to (508.29, 535.33, 180) mm, rotated rx -180 ry 0 rz 160 deg; joints [10.437, 52.949, -3.579, -142.253, 55.845, 156.507]
  Set speed (17.7 mm/s)
  Call Extruder(236.65280)
  MoveL 9994 to (506.79, 535.65, 180) mm, rotated rx 180 ry 0 rz 160 deg; joints [10.509, 52.697, -3.111, -142.263, 56.045, 156.623]
  Set speed (17.7 mm/s)
  Call Extruder(241.43385)
  MoveL 9995 to (505.31, 535.9, 180) mm, rotated rx 180 ry 0 rz 160 deg; joints [10.573, 52.448, -2.646, -142.28, 56.241, 156.742]
  Set speed (17.7 mm/s)
  Call Extruder(245.98535)
  MoveL 9996 to (503.9, 536.08, 180) mm, rotated rx -180 ry 0 rz 160 deg; joints [10.627, 52.209, -2.201, -142.304, 56.425, 156.86]
  Set speed (17.7 mm/s)
  Call Extruder(250.85093)
  MoveL 9997 to (502.38, 536.21, 180) mm, rotated rx -180 ry 0 rz 160 deg; joints [10.678, 51.951, -1.721, -142.338, 56.621, 156.992]
  Set speed (17.7 mm/s)
  Call Extruder(255.64675)
  MoveL 9998 to (500.87, 536.27, 180) mm, rotated rx 180 ry 0 rz 160 deg; joints [10.721, 51.696, -1.246, -142.379, 56.812, 157.126]
  Set speed (17.7 mm/s)
  Call Extruder(260.28593)
  MoveL 9999 to (499.42, 536.28, 180) mm, rotated rx -180 ry 0 rz 160 deg; joints [10.756, 51.448, -0.785, -142.425, 56.994, 157.261]
  Set speed (10.0 mm/s)
  MoveL 10000 to (499.42, 536.28, 184) mm, rotated rx 180 ry 0 rz 160 deg; joints [10.756, 50.917, -0.731, -142.234, 56.616, 156.912]
  Set speed (120.0 mm/s)
  MoveL 10001 to (499.43, 535.65, 184) mm, rotated rx 180 ry 0 rz 160 deg; joints [10.678, 50.899, -0.698, -142.327, 56.598, 156.971]
  Set speed (17.9 mm/s)
  Call Extruder(264.97054)
  MoveL 10002 to (497.95, 535.59, 184) mm, rotated rx 180 ry 0 rz 160 deg; joints [10.705, 50.645, -0.228, -142.383, 56.779, 157.112]
  Set speed (17.9 mm/s)
  Call Extruder(269.60294)
  MoveL 10003 to (496.49, 535.48, 184) mm, rotated rx 180 ry 0 rz 160 deg; joints [10.726, 50.393, 0.237, -142.446, 56.956, 157.255]
  Set speed (17.9 mm/s)
  Call Extruder(274.14567)
  MoveL 10004 to (495.06, 535.31, 184) mm, rotated rx 180 ry 0 rz 160 deg; joints [10.738, 50.146, 0.693, -142.514, 57.127, 157.399]
  Set speed (17.9 mm/s)
  Call Extruder(278.73940)
  MoveL 10005 to (493.63, 535.08, 184) mm, rotated rx -180 ry 0 rz 160 deg; joints [10.743, 49.897, 1.152, -142.591, 57.296, 157.548]
  Set speed (17.9 mm/s)
  Call Extruder(283.45829)
  MoveL 10006 to (492.17, 534.78, 184) mm, rotated rx -180 ry 0 rz 160 deg; joints [10.741, 49.643, 1.622, -142.677, 57.466, 157.705]
  Set speed (17.8 mm/s)
  Call Extruder(287.91637)
  MoveL 10007 to (490.8, 534.44, 184) mm, rotated rx 180 ry 0 rz 160 deg; joints [10.731, 49.404, 2.062, -142.766, 57.622, 157.855]
  Call Extruder(292.43875)
  MoveL 10008 to (489.42, 534.05, 184) mm, rotated rx -180 ry 0 rz 160 deg; joints [10.714, 49.163, 2.506, -142.862, 57.778, 158.011]
  Call Extruder(297.12342)
  MoveL 10009 to (488.02, 533.58, 184) mm, rotated rx -180 ry 0 rz 160 deg; joints [10.688, 48.916, 2.961, -142.969, 57.934, 158.174]
  Call Extruder(301.69930)
  MoveL 10010 to (486.66, 533.06, 184) mm, rotated rx -180 ry 0 rz 160 deg; joints [10.655, 48.677, 3.401, -143.081, 58.083, 158.336]
  Set speed (17.8 mm/s)
  Call Extruder(304.14264)
  MoveL 10011 to (485.95, 532.77, 184) mm, rotated rx -180 ry 0 rz 160 deg; joints [10.635, 48.551, 3.633, -143.142, 58.16, 158.422]
  Set speed (17.8 mm/s)
  Call Extruder(306.26411)
  MoveL 10012 to (485.34, 532.5, 184) mm, rotated rx -180 ry 0 rz 160 deg; joints [10.615, 48.443, 3.834, -143.198, 58.226, 158.498]
  Set speed (17.9 mm/s)
  Call Extruder(308.67544)
  MoveL 10013 to (484.65, 532.18, 184) mm, rotated rx 180 ry 0 rz 160 deg; joints [10.591, 48.32, 4.06, -143.264, 58.3, 158.585]
  Set speed (17.8 mm/s)
  Call Extruder(311.84583)
  MoveL 10014 to (483.75, 531.74, 184) mm, rotated rx -180 ry 0 rz 160 deg; joints [10.556, 48.16, 4.355, -143.351, 58.395, 158.7]
  Set speed (17.8 mm/s)
  Call Extruder(315.78260)
  MoveL 10015 to (482.65, 531.15, 184) mm, rotated rx -180 ry 0 rz 160 deg; joints [10.506, 47.963, 4.716, -143.466, 58.51, 158.843]
  Set speed (17.9 mm/s)
  Call Extruder(320.18324)
  MoveL 10016 to (481.45, 530.45, 184) mm, rotated rx -180 ry 0 rz 160 deg; joints [10.445, 47.748, 5.113, -143.599, 58.633, 159.005]
  Set speed (17.9 mm/s)
  Call Extruder(322.46655)
  MoveL 10017 to (480.84, 530.06, 184) mm, rotated rx 180 ry 0 rz 160 deg; joints [10.41, 47.637, 5.316, -143.67, 58.696, 159.089]
  Call Extruder(324.84099)
  MoveL 10018 to (480.21, 529.65, 184) mm, rotated rx -180 ry 0 rz 160 deg; joints [10.372, 47.523, 5.525, -143.746, 58.759, 159.176]
  Set speed (17.9 mm/s)
  Call Extruder(329.35932)
  MoveL 10019 to (479.03, 528.83, 184) mm, rotated rx 180 ry 0 rz 160 deg; joints [10.294, 47.31, 5.917, -143.895, 58.875, 159.344]
  Set speed (17.9 mm/s)
  Call Extruder(331.69790)
  MoveL 10020 to (478.44, 528.39, 184) mm, rotated rx -180 ry 0 rz 160 deg; joints [10.251, 47.202, 6.116, -143.975, 58.934, 159.43]
  Set speed (17.9 mm/s)
  Call Extruder(334.05668)
  MoveL 10021 to (477.85, 527.94, 184) mm, rotated rx -180 ry 0 rz 160 deg; joints [10.205, 47.094, 6.314, -144.056, 58.991, 159.518]
  Call Extruder(338.78130)
  MoveL 10022 to (476.7, 526.98, 184) mm, rotated rx 180 ry 0 rz 160 deg; joints [10.108, 46.883, 6.703, -144.225, 59.1, 159.694]
  Set speed (17.9 mm/s)
  Call Extruder(343.21980)
  MoveL 10023 to (475.65, 526.05, 184) mm, rotated rx 180 ry 0 rz 160 deg; joints [10.01, 46.689, 7.057, -144.388, 59.198, 159.859]
  Set speed (17.9 mm/s)
  Call Extruder(345.59344)
  MoveL 10024 to (475.11, 525.53, 184) mm, rotated rx 180 ry 0 rz 160 deg; joints [9.954, 46.588, 7.243, -144.478, 59.247, 159.947]
  Set speed (17.9 mm/s)
  Call Extruder(347.90268)
  MoveL 10025 to (474.59, 525.01, 184) mm, rotated rx 180 ry 0 rz 160 deg; joints [9.899, 46.492, 7.42, -144.567, 59.294, 160.032]
  Set speed (17.8 mm/s)
  Call Extruder(350.16001)
  MoveL 10026 to (474.1, 524.5, 184) mm, rotated rx -180 ry 0 rz 160 deg; joints [9.843, 46.399, 7.59, -144.655, 59.338, 160.116]
  Set speed (17.8 mm/s)
  Call Extruder(352.53567)
  MoveL 10027 to (473.59, 523.95, 184) mm, rotated rx 180 ry 0 rz 160 deg; joints [9.782, 46.303, 7.766, -144.749, 59.382, 160.203]
  Set speed (17.8 mm/s)
  Call Extruder(356.96160)
  MoveL 10028 to (472.67, 522.89, 184) mm, rotated rx -180 ry 0 rz 160 deg; joints [9.663, 46.129, 8.086, -144.928, 59.462, 160.366]
  Set speed (17.9 mm/s)
  Call Extruder(359.42549)
  MoveL 10029 to (472.17, 522.29, 184) mm, rotated rx -180 ry 0 rz 160 deg; joints [9.595, 46.035, 8.259, -145.029, 59.503, 160.457]
  Set speed (17.9 mm/s)
  Call Extruder(361.68941)
  MoveL 10030 to (471.73, 521.73, 184) mm, rotated rx -180 ry 0 rz 160 deg; joints [9.53, 45.95, 8.414, -145.124, 59.539, 160.54]
  Set speed (17.9 mm/s)
  Call Extruder(366.25453)
  MoveL 10031 to (470.88, 520.56, 184) mm, rotated rx 180 ry 0 rz 160 deg; joints [9.395, 45.784, 8.718, -145.318, 59.608, 160.706]
  Set speed (17.9 mm/s)
  Call Extruder(368.70290)
  MoveL 10032 to (470.43, 519.92, 184) mm, rotated rx 180 ry 0 rz 160 deg; joints [9.32, 45.698, 8.875, -145.424, 59.642, 160.794]
  Set speed (17.9 mm/s)
  Call Extruder(373.31550)
  MoveL 10033 to (469.64, 518.7, 184) mm, rotated rx -180 ry 0 rz 160 deg; joints [9.174, 45.543, 9.16, -145.627, 59.701, 160.96]
  Call Extruder(375.55851)
  MoveL 10034 to (469.28, 518.09, 184) mm, rotated rx -180 ry 0 rz 160 deg; joints [9.1, 45.47, 9.293, -145.727, 59.726, 161.04]
  Set speed (17.9 mm/s)
  Call Extruder(377.93159)
  MoveL 10035 to (468.91, 517.44, 184) mm, rotated rx 180 ry 0 rz 160 deg; joints [9.022, 45.396, 9.43, -145.834, 59.752, 161.124]
  Set speed (17.8 mm/s)
  Call Extruder(382.43266)
  MoveL 10036 to (468.23, 516.18, 184) mm, rotated rx -180 ry 0 rz 160 deg; joints [8.868, 45.259, 9.679, -146.039, 59.797, 161.282]
  Set speed (17.8 mm/s)
  Call Extruder(384.75181)
  MoveL 10037 to (467.91, 515.53, 184) mm, rotated rx -180 ry 0 rz 160 deg; joints [8.787, 45.192, 9.802, -146.146, 59.817, 161.363]
  Set speed (17.9 mm/s)
  Call Extruder(389.37164)
  MoveL 10038 to (467.3, 514.2, 184) mm, rotated rx 180 ry 0 rz 160 deg; joints [8.621, 45.066, 10.034, -146.362, 59.852, 161.522]
  Set speed (17.9 mm/s)
  Call Extruder(393.87534)
  MoveL 10039 to (466.76, 512.88, 184) mm, rotated rx 180 ry 0 rz 160 deg; joints [8.454, 44.951, 10.244, -146.576, 59.878, 161.675]
  Set speed (17.8 mm/s)
  Call Extruder(395.90647)
  MoveL 10040 to (466.53, 512.28, 184) mm, rotated rx 180 ry 0 rz 160 deg; joints [8.377, 44.902, 10.334, -146.673, 59.888, 161.743]
  Set speed (17.8 mm/s)
  Call Extruder(398.77974)
  MoveL 10041 to (466.23, 511.42, 184) mm, rotated rx -180 ry 0 rz 160 deg; joints [8.268, 44.835, 10.456, -146.81, 59.901, 161.838]
  Set speed (17.8 mm/s)
  Call Extruder(403.14286)
  MoveL 10042 to (465.81, 510.11, 184) mm, rotated rx -180 ry 0 rz 160 deg; joints [8.098, 44.74, 10.629, -147.022, 59.914, 161.981]
  Set speed (17.9 mm/s)
  Call Extruder(407.75450)
  MoveL 10043 to (465.42, 508.7, 184) mm, rotated rx -180 ry 0 rz 160 deg; joints [7.915, 44.65, 10.795, -147.247, 59.92, 162.129]
  Call Extruder(412.37663)
  MoveL 10044 to (465.1, 507.28, 184) mm, rotated rx 180 ry 0 rz 160 deg; joints [7.728, 44.569, 10.943, -147.474, 59.92, 162.274]
  Set speed (17.9 mm/s)
  Call Extruder(417.13779)
  MoveL 10045 to (464.82, 505.79, 184) mm, rotated rx 180 ry 0 rz 160 deg; joints [7.532, 44.495, 11.077, -147.709, 59.911, 162.42]
  Call Extruder(421.76161)
  MoveL 10046 to (464.61, 504.35, 184) mm, rotated rx 180 ry 0 rz 160 deg; joints [7.338, 44.434, 11.19, -147.937, 59.896, 162.559]
  Set speed (17.9 mm/s)
  Call Extruder(426.36071)
  MoveL 10047 to (464.46, 502.9, 184) mm, rotated rx -180 ry 0 rz 160 deg; joints [7.144, 44.382, 11.285, -148.165, 59.875, 162.693]
  Call Extruder(431.14591)
  MoveL 10048 to (464.38, 501.39, 184) mm, rotated rx -180 ry 0 rz 160 deg; joints [6.939, 44.339, 11.363, -148.402, 59.844, 162.827]
  Set speed (17.8 mm/s)
  Call Extruder(435.50244)
  MoveL 10049 to (464.35, 500.01, 184) mm, rotated rx 180 ry 0 rz 160 deg; joints [6.752, 44.31, 11.416, -148.617, 59.81, 162.946]
  Call Extruder(439.72915)
  MoveL 10050 to (464.37, 498.67, 184) mm, rotated rx -180 ry 0 rz 160 deg; joints [6.569, 44.289, 11.455, -148.824, 59.771, 163.059]
  Set speed (17.8 mm/s)
  Call Extruder(443.72562)
  MoveL 10051 to (464.44, 497.41, 184) mm, rotated rx 180 ry 0 rz 160 deg; joints [6.395, 44.277, 11.476, -149.02, 59.729, 163.161]
  Set speed (17.9 mm/s)
  Call Extruder(447.93139)
  MoveL 10052 to (464.56, 496.09, 184) mm, rotated rx -180 ry 0 rz 160 deg; joints [6.212, 44.273, 11.483, -149.224, 59.678, 163.266]
  Set speed (17.9 mm/s)
  Call Extruder(452.08277)
  MoveL 10053 to (464.73, 494.79, 184) mm, rotated rx -180 ry 0 rz 160 deg; joints [6.031, 44.278, 11.474, -149.423, 59.623, 163.365]
  Set speed (17.9 mm/s)
  Call Extruder(456.32732)
  MoveL 10054 to (464.95, 493.46, 184) mm, rotated rx -180 ry 0 rz 160 deg; joints [5.847, 44.291, 11.451, -149.625, 59.562, 163.462]
  Call Extruder(460.32794)
  MoveL 10055 to (465.21, 492.22, 184) mm, rotated rx -180 ry 0 rz 160 deg; joints [5.673, 44.311, 11.414, -149.813, 59.498, 163.55]
  Set speed (17.9 mm/s)
  Call Extruder(464.53746)
  MoveL 10056 to (465.52, 490.93, 184) mm, rotated rx -180 ry 0 rz 160 deg; joints [5.492, 44.34, 11.361, -150.008, 59.426, 163.639]
  Call Extruder(468.61475)
  MoveL 10057 to (465.88, 489.69, 184) mm, rotated rx -180 ry 0 rz 160 deg; joints [5.318, 44.377, 11.294, -150.193, 59.351, 163.72]
  Call Extruder(472.76601)
  MoveL 10058 to (466.28, 488.44, 184) mm, rotated rx -180 ry 0 rz 160 deg; joints [5.142, 44.422, 11.212, -150.379, 59.269, 163.799]
  Call Extruder(477.01248)
  MoveL 10059 to (466.74, 487.17, 184) mm, rotated rx -180 ry 0 rz 160 deg; joints [4.963, 44.476, 11.113, -150.565, 59.181, 163.875]
  Set speed (17.8 mm/s)
  Call Extruder(480.32614)
  MoveL 10060 to (467.13, 486.2, 184) mm, rotated rx 180 ry 0 rz 160 deg; joints [4.826, 44.523, 11.026, -150.707, 59.108, 163.932]
  Set speed (17.8 mm/s)
  Call Extruder(485.22167)
  MoveL 10061 to (467.76, 484.79, 184) mm, rotated rx 180 ry 0 rz 160 deg; joints [4.626, 44.604, 10.879, -150.912, 58.995, 164.009]
  Set speed (17.9 mm/s)
  Call Extruder(489.38687)
  MoveL 10062 to (468.34, 483.61, 184) mm, rotated rx 180 ry 0 rz 160 deg; joints [4.459, 44.68, 10.738, -151.081, 58.893, 164.07]
  Call Extruder(493.58810)
  MoveL 10063 to (468.97, 482.44, 184) mm, rotated rx 180 ry 0 rz 160 deg; joints [4.293, 44.765, 10.583, -151.247, 58.786, 164.127]
  Call Extruder(497.80905)
  MoveL 10064 to (469.65, 481.29, 184) mm, rotated rx -180 ry 0 rz 160 deg; joints [4.129, 44.859, 10.412, -151.408, 58.673, 164.179]
  Set speed (17.9 mm/s)
  Call Extruder(501.87815)
  MoveL 10065 to (470.35, 480.21, 184) mm, rotated rx 180 ry 0 rz 160 deg; joints [3.975, 44.956, 10.234, -151.558, 58.561, 164.224]
  Set speed (17.9 mm/s)
  Call Extruder(506.03256)
  MoveL 10066 to (471.1, 479.13, 184) mm, rotated rx -180 ry 0 rz 160 deg; joints [3.822, 45.062, 10.04, -151.706, 58.441, 164.265]
  Call Extruder(510.26193)
  MoveL 10067 to (471.9, 478.06, 184) mm, rotated rx 180 ry 0 rz 160 deg; joints [3.67, 45.178, 9.828, -151.85, 58.315, 164.302]
  Set speed (17.9 mm/s)
  Call Extruder(514.28171)
  MoveL 10068 to (472.7, 477.07, 184) mm, rotated rx -180 ry 0 rz 160 deg; joints [3.529, 45.295, 9.614, -151.981, 58.192, 164.332]
  Set speed (17.9 mm/s)
  Call Extruder(518.47730)
  MoveL 10069 to (473.58, 476.07, 184) mm, rotated rx -180 ry 0 rz 160 deg; joints [3.387, 45.423, 9.38, -152.111, 58.059, 164.359]
  Set speed (17.9 mm/s)
  Call Extruder(522.70628)
  MoveL 10070 to (474.49, 475.09, 184) mm, rotated rx 180 ry 0 rz 160 deg; joints [3.248, 45.559, 9.13, -152.236, 57.921, 164.38]
  Set speed (17.9 mm/s)
  Call Extruder(526.75623)
  MoveL 10071 to (475.4, 474.19, 184) mm, rotated rx -180 ry 0 rz 160 deg; joints [3.12, 45.696, 8.879, -152.348, 57.786, 164.395]
  Call Extruder(530.96207)
  MoveL 10072 to (476.39, 473.29, 184) mm, rotated rx -180 ry 0 rz 160 deg; joints [2.992, 45.845, 8.606, -152.458, 57.642, 164.405]
  Call Extruder(535.11007)
  MoveL 10073 to (477.38, 472.44, 184) mm, rotated rx -180 ry 0 rz 160 deg; joints [2.871, 45.997, 8.327, -152.558, 57.497, 164.409]
  Set speed (17.9 mm/s)
  Call Extruder(539.13652)
  MoveL 10074 to (478.38, 471.65, 184) mm, rotated rx 180 ry 0 rz 160 deg; joints [2.759, 46.151, 8.045, -152.649, 57.353, 164.408]
  Set speed (17.8 mm/s)
  Call Extruder(541.33840)
  MoveL 10075 to (478.94, 471.23, 184) mm, rotated rx -180 ry 0 rz 160 deg; joints [2.699, 46.236, 7.889, -152.697, 57.274, 164.407]
  Call Extruder(543.26472)
  MoveL 10076 to (479.43, 470.88, 184) mm, rotated rx -180 ry 0 rz 160 deg; joints [2.649, 46.313, 7.747, -152.735, 57.203, 164.402]
  Set speed (17.9 mm/s)
  Call Extruder(547.55692)
  MoveL 10077 to (480.56, 470.12, 184) mm, rotated rx -180 ry 0 rz 160 deg; joints [2.541, 46.489, 7.426, -152.816, 57.044, 164.39]
  Call Extruder(551.71516)
  MoveL 10078 to (481.67, 469.42, 184) mm, rotated rx 180 ry 0 rz 160 deg; joints [2.442, 46.664, 7.104, -152.886, 56.887, 164.372]
  Set speed (17.8 mm/s)
  Call Extruder(555.63608)
  MoveL 10079 to (482.75, 468.8, 184) mm, rotated rx 180 ry 0 rz 160 deg; joints [2.354, 46.833, 6.793, -152.945, 56.737, 164.351]
  Call Extruder(560.00341)
  MoveL 10080 to (483.97, 468.16, 184) mm, rotated rx -180 ry 0 rz 160 deg; joints [2.262, 47.027, 6.437, -153.002, 56.567, 164.321]
  Set speed (17.9 mm/s)
  Call Extruder(564.16068)
  MoveL 10081 to (485.15, 467.59, 184) mm, rotated rx -180 ry 0 rz 160 deg; joints [2.181, 47.217, 6.088, -153.048, 56.404, 164.286]
  Call Extruder(568.35389)
  MoveL 10082 to (486.37, 467.06, 184) mm, rotated rx -180 ry 0 rz 160 deg; joints [2.105, 47.412, 5.73, -153.087, 56.238, 164.246]
  Set speed (17.8 mm/s)
  Call Extruder(572.35387)
  MoveL 10083 to (487.55, 466.6, 184) mm, rotated rx 180 ry 0 rz 160 deg; joints [2.039, 47.602, 5.38, -153.115, 56.078, 164.201]
  Set speed (17.8 mm/s)
  Call Extruder(576.43176)
  MoveL 10084 to (488.76, 466.17, 184) mm, rotated rx -180 ry 0 rz 160 deg; joints [1.977, 47.8, 5.017, -153.136, 55.913, 164.151]
  Set speed (17.8 mm/s)
  Call Extruder(580.77125)
  MoveL 10085 to (490.07, 465.76, 184) mm, rotated rx -180 ry 0 rz 160 deg; joints [1.918, 48.013, 4.624, -153.149, 55.737, 164.092]
  Set speed (17.9 mm/s)
  Call Extruder(584.94842)
  MoveL 10086 to (491.35, 465.41, 184) mm, rotated rx -180 ry 0 rz 160 deg; joints [1.868, 48.223, 4.238, -153.154, 55.566, 164.029]
  Set speed (17.9 mm/s)
  Call Extruder(589.01132)
  MoveL 10087 to (492.6, 465.12, 184) mm, rotated rx 180 ry 0 rz 160 deg; joints [1.825, 48.429, 3.858, -153.15, 55.399, 163.962]
  Set speed (17.8 mm/s)
  Call Extruder(593.13163)
  MoveL 10088 to (493.88, 464.88, 184) mm, rotated rx 180 ry 0 rz 160 deg; joints [1.788, 48.641, 3.468, -153.137, 55.23, 163.888]
  Set speed (17.8 mm/s)
  Call Extruder(596.99287)
  MoveL 10089 to (495.09, 464.69, 184) mm, rotated rx -180 ry 0 rz 160 deg; joints [1.759, 48.842, 3.098, -153.118, 55.071, 163.815]
  Call Extruder(601.51797)
  MoveL 10090 to (496.51, 464.52, 184) mm, rotated rx 180 ry 0 rz 160 deg; joints [1.732, 49.08, 2.66, -153.086, 54.885, 163.722]
  Set speed (17.8 mm/s)
  Call Extruder(605.62312)
  MoveL 10091 to (497.8, 464.42, 184) mm, rotated rx 180 ry 0 rz 160 deg; joints [1.713, 49.298, 2.258, -153.049, 54.716, 163.633]
  Set speed (17.9 mm/s)
  Call Extruder(609.85695)
  MoveL 10092 to (499.14, 464.36, 184) mm, rotated rx -180 ry 0 rz 160 deg; joints [1.701, 49.524, 1.841, -153.002, 54.542, 163.535]
  Set speed (17.9 mm/s)
  Call Extruder(613.92652)
  MoveL 10093 to (500.43, 464.35, 184) mm, rotated rx -180 ry 0 rz 160 deg; joints [1.695, 49.743, 1.437, -152.949, 54.376, 163.436]
  Set speed (17.9 mm/s)
  Call Extruder(618.14158)
  MoveL 10094 to (501.76, 464.39, 184) mm, rotated rx -180 ry 0 rz 160 deg; joints [1.695, 49.971, 1.017, -152.886, 54.204, 163.328]
  Set speed (17.9 mm/s)
  Call Extruder(622.23236)
  MoveL 10095 to (503.05, 464.48, 184) mm, rotated rx -180 ry 0 rz 160 deg; joints [1.702, 50.193, 0.607, -152.817, 54.039, 163.218]
  Set speed (17.9 mm/s)
  Call Extruder(626.45085)
  MoveL 10096 to (504.38, 464.62, 184) mm, rotated rx -180 ry 0 rz 160 deg; joints [1.714, 50.422, 0.184, -152.737, 53.87, 163.099]
  Call Extruder(630.74250)
  MoveL 10097 to (505.72, 464.81, 184) mm, rotated rx -180 ry 0 rz 160 deg; joints [1.733, 50.655, -0.247, -152.648, 53.7, 162.973]
  Set speed (17.9 mm/s)
  Call Extruder(634.72957)
  MoveL 10098 to (506.97, 465.04, 184) mm, rotated rx 180 ry 0 rz 160 deg; joints [1.757, 50.872, -0.647, -152.558, 53.544, 162.852]
  Call Extruder(638.82755)
  MoveL 10099 to (508.23, 465.31, 184) mm, rotated rx -180 ry 0 rz 160 deg; joints [1.786, 51.094, -1.058, -152.458, 53.385, 162.723]
  Set speed (17.9 mm/s)
  Call Extruder(642.88214)
  MoveL 10100 to (509.48, 465.63, 184) mm, rotated rx 180 ry 0 rz 160 deg; joints [1.821, 51.313, -1.464, -152.352, 53.231, 162.59]
  Set speed (17.9 mm/s)
  Call Extruder(647.11035)
  MoveL 10101 to (510.76, 466.01, 184) mm, rotated rx -180 ry 0 rz 160 deg; joints [1.863, 51.541, -1.885, -152.235, 53.072, 162.448]
  Set speed (17.9 mm/s)
  Call Extruder(651.32293)
  MoveL 10102 to (512.02, 466.44, 184) mm, rotated rx -180 ry 0 rz 160 deg; joints [1.911, 51.767, -2.302, -152.11, 52.917, 162.301]
  Set speed (17.9 mm/s)
  Call Extruder(655.42148)
  MoveL 10103 to (513.24, 466.9, 184) mm, rotated rx -180 ry 0 rz 160 deg; joints [1.963, 51.985, -2.706, -151.982, 52.769, 162.155]
  Set speed (17.9 mm/s)
  Call Extruder(659.61714)
  MoveL 10104 to (514.46, 467.41, 184) mm, rotated rx 180 ry 0 rz 160 deg; joints [2.022, 52.206, -3.115, -151.845, 52.621, 162.001]
  Set speed (17.9 mm/s)
  Call Extruder(663.76950)
  MoveL 10105 to (515.65, 467.97, 184) mm, rotated rx -180 ry 0 rz 160 deg; joints [2.085, 52.423, -3.516, -151.703, 52.478, 161.845]
  Set speed (17.9 mm/s)
  Call Extruder(667.77506)
  MoveL 10106 to (516.78, 468.54, 184) mm, rotated rx 180 ry 0 rz 160 deg; joints [2.151, 52.629, -3.899, -151.559, 52.344, 161.691]
  Set speed (17.9 mm/s)
  Call Extruder(672.05133)
  MoveL 10107 to (517.96, 469.2, 184) mm, rotated rx -180 ry 0 rz 160 deg; joints [2.226, 52.847, -4.302, -151.4, 52.205, 161.524]
  Set speed (17.9 mm/s)
  Call Extruder(676.11749)
  MoveL 10108 to (519.06, 469.87, 184) mm, rotated rx -180 ry 0 rz 160 deg; joints [2.302, 53.051, -4.68, -151.244, 52.076, 161.362]
  Set speed (17.9 mm/s)
  Call Extruder(680.35624)
  MoveL 10109 to (520.18, 470.61, 184) mm, rotated rx 180 ry 0 rz 160 deg; joints [2.387, 53.26, -5.068, -151.075, 51.947, 161.19]
  Set speed (17.9 mm/s)
  Call Extruder(684.41810)
  MoveL 10110 to (521.23, 471.36, 184) mm, rotated rx 180 ry 0 rz 160 deg; joints [2.472, 53.458, -5.434, -150.908, 51.827, 161.023]
  Set speed (17.9 mm/s)
  Call Extruder(688.60831)
  MoveL 10111 to (522.28, 472.17, 184) mm, rotated rx 180 ry 0 rz 160 deg; joints [2.565, 53.657, -5.803, -150.731, 51.709, 160.848]
  Set speed (17.9 mm/s)
  Call Extruder(692.75080)
  MoveL 10112 to (523.29, 473, 184) mm, rotated rx 180 ry 0 rz 160 deg; joints [2.661, 53.85, -6.161, -150.552, 51.597, 160.674]
  Set speed (17.9 mm/s)
  Call Extruder(696.80206)
  MoveL 10113 to (524.24, 473.86, 184) mm, rotated rx -180 ry 0 rz 160 deg; joints [2.759, 54.034, -6.503, -150.372, 51.492, 160.501]
  Set speed (17.9 mm/s)
  Call Extruder(701.08132)
  MoveL 10114 to (525.22, 474.8, 184) mm, rotated rx 180 ry 0 rz 160 deg; joints [2.866, 54.224, -6.856, -150.179, 51.387, 160.317]
  Call Extruder(705.50591)
  MoveL 10115 to (526.19, 475.81, 184) mm, rotated rx -180 ry 0 rz 160 deg; joints [2.982, 54.415, -7.209, -149.974, 51.285, 160.126]
  Set speed (17.9 mm/s)
  Call Extruder(707.91594)
  MoveL 10116 to (526.7, 476.37, 184) mm, rotated rx 180 ry 0 rz 160 deg; joints [3.046, 54.516, -7.397, -149.861, 51.232, 160.022]
  Call Extruder(710.23255)
  MoveL 10117 to (527.18, 476.93, 184) mm, rotated rx 180 ry 0 rz 160 deg; joints [3.11, 54.612, -7.575, -149.752, 51.183, 159.921]
  Set speed (17.9 mm/s)
  Call Extruder(712.53277)
  MoveL 10118 to (527.64, 477.49, 184) mm, rotated rx 180 ry 0 rz 160 deg; joints [3.174, 54.705, -7.747, -149.642, 51.136, 159.821]
  Call Extruder(714.86624)
  MoveL 10119 to (528.11, 478.06, 184) mm, rotated rx -180 ry 0 rz 160 deg; joints [3.24, 54.798, -7.92, -149.53, 51.09, 159.719]
  Call Extruder(717.10396)
  MoveL 10120 to (528.54, 478.63, 184) mm, rotated rx 180 ry 0 rz 160 deg; joints [3.304, 54.885, -8.082, -149.422, 51.048, 159.622]
  Set speed (17.9 mm/s)
  Call Extruder(719.38323)
  MoveL 10121 to (528.96, 479.21, 184) mm, rotated rx 180 ry 0 rz 160 deg; joints [3.371, 54.972, -8.244, -149.311, 51.007, 159.522]
  Set speed (17.9 mm/s)
  Call Extruder(721.70258)
  MoveL 10122 to (529.38, 479.81, 184) mm, rotated rx 180 ry 0 rz 160 deg; joints [3.439, 55.058, -8.404, -149.198, 50.968, 159.421]
  Call Extruder(723.97751)
  MoveL 10123 to (529.78, 480.41, 184) mm, rotated rx -180 ry 0 rz 160 deg; joints [3.508, 55.142, -8.559, -149.086, 50.93, 159.323]
  Set speed (17.9 mm/s)
  Call Extruder(726.36103)
  MoveL 10124 to (530.19, 481.04, 184) mm, rotated rx 180 ry 0 rz 160 deg; joints [3.58, 55.226, -8.716, -148.968, 50.894, 159.219]
  Set speed (17.9 mm/s)
  Call Extruder(728.69954)
  MoveL 10125 to (530.58, 481.67, 184) mm, rotated rx 180 ry 0 rz 160 deg; joints [3.652, 55.307, -8.867, -148.852, 50.86, 159.118]
  Set speed (17.9 mm/s)
  Call Extruder(733.17704)
  MoveL 10126 to (531.28, 482.9, 184) mm, rotated rx 180 ry 0 rz 160 deg; joints [3.793, 55.457, -9.145, -148.628, 50.8, 158.925]
  Call Extruder(735.59457)
  MoveL 10127 to (531.64, 483.58, 184) mm, rotated rx -180 ry 0 rz 160 deg; joints [3.87, 55.535, -9.289, -148.507, 50.771, 158.821]
  Set speed (17.9 mm/s)
  Call Extruder(738.55314)
  MoveL 10128 to (532.06, 484.41, 184) mm, rotated rx 180 ry 0 rz 160 deg; joints [3.966, 55.626, -9.459, -148.358, 50.739, 158.696]
  Set speed (17.9 mm/s)
  Call Extruder(742.36262)
  MoveL 10129 to (532.57, 485.51, 184) mm, rotated rx 180 ry 0 rz 160 deg; joints [4.091, 55.739, -9.668, -148.166, 50.703, 158.535]
  Set speed (17.9 mm/s)
  Call Extruder(746.92516)
  MoveL 10130 to (533.13, 486.84, 184) mm, rotated rx 180 ry 0 rz 160 deg; joints [4.243, 55.866, -9.904, -147.935, 50.666, 158.344]
  Call Extruder(751.71780)
  MoveL 10131 to (533.66, 488.26, 184) mm, rotated rx 180 ry 0 rz 160 deg; joints [4.406, 55.989, -10.133, -147.694, 50.637, 158.147]
  Set speed (17.9 mm/s)
  Call Extruder(756.24963)
  MoveL 10132 to (534.11, 489.62, 184) mm, rotated rx 180 ry 0 rz 160 deg; joints [4.563, 56.096, -10.332, -147.465, 50.618, 157.964]
  Set speed (17.9 mm/s)
  Call Extruder(760.75156)
  MoveL 10133 to (534.49, 490.99, 184) mm, rotated rx 180 ry 0 rz 160 deg; joints [4.721, 56.192, -10.511, -147.24, 50.608, 157.786]
  Set speed (17.9 mm/s)
  Call Extruder(765.45324)
  MoveL 10134 to (534.84, 492.44, 184) mm, rotated rx -180 ry 0 rz 160 deg; joints [4.887, 56.283, -10.681, -147.005, 50.605, 157.605]
  Set speed (17.9 mm/s)
  Call Extruder(770.13682)
  MoveL 10135 to (535.12, 493.89, 184) mm, rotated rx -180 ry 0 rz 160 deg; joints [5.055, 56.363, -10.829, -146.774, 50.612, 157.429]
  Set speed (17.9 mm/s)
  Call Extruder(774.65900)
  MoveL 10136 to (535.34, 495.31, 184) mm, rotated rx -180 ry 0 rz 160 deg; joints [5.219, 56.431, -10.954, -146.552, 50.626, 157.264]
  Call Extruder(779.43892)
  MoveL 10137 to (535.51, 496.81, 184) mm, rotated rx 180 ry 0 rz 160 deg; joints [5.393, 56.49, -11.066, -146.321, 50.651, 157.095]
  Set speed (17.9 mm/s)
  Call Extruder(783.95932)
  MoveL 10138 to (535.61, 498.24, 184) mm, rotated rx -180 ry 0 rz 160 deg; joints [5.559, 56.537, -11.152, -146.105, 50.683, 156.941]
  Set speed (17.9 mm/s)
  Call Extruder(788.57028)
  MoveL 10139 to (535.65, 499.69, 184) mm, rotated rx -180 ry 0 rz 160 deg; joints [5.729, 56.573, -11.22, -145.889, 50.724, 156.79]
  Set speed (17.9 mm/s)
  Call Extruder(793.07935)
  MoveL 10140 to (535.63, 501.12, 184) mm, rotated rx 180 ry 0 rz 160 deg; joints [5.896, 56.598, -11.266, -145.681, 50.772, 156.65]
  Set speed (17.9 mm/s)
  Call Extruder(797.77819)
  MoveL 10141 to (535.56, 502.61, 184) mm, rotated rx 180 ry 0 rz 160 deg; joints [6.071, 56.614, -11.296, -145.468, 50.83, 156.509]
  Call Extruder(802.39089)
  MoveL 10142 to (535.42, 504.06, 184) mm, rotated rx 180 ry 0 rz 160 deg; joints [6.242, 56.617, -11.302, -145.264, 50.896, 156.379]
  Set speed (17.9 mm/s)
  Call Extruder(807.09489)
  MoveL 10143 to (535.22, 505.54, 184) mm, rotated rx 180 ry 0 rz 160 deg; joints [6.417, 56.611, -11.289, -145.06, 50.971, 156.253]
  Set speed (17.9 mm/s)
  Call Extruder(811.59712)
  MoveL 10144 to (534.97, 506.94, 184) mm, rotated rx -180 ry 0 rz 160 deg; joints [6.584, 56.593, -11.257, -144.871, 51.051, 156.141]
  Set speed (17.9 mm/s)
  Call Extruder(816.38603)
  MoveL 10145 to (534.64, 508.42, 184) mm, rotated rx 180 ry 0 rz 160 deg; joints [6.761, 56.563, -11.201, -144.674, 51.144, 156.029]
  Set speed (17.9 mm/s)
  Call Extruder(820.64679)
  MoveL 10146 to (534.3, 509.72, 184) mm, rotated rx -180 ry 0 rz 160 deg; joints [6.919, 56.527, -11.133, -144.505, 51.233, 155.937]
  Set speed (17.9 mm/s)
  Call Extruder(825.27409)
  MoveL 10147 to (533.87, 511.12, 184) mm, rotated rx -180 ry 0 rz 160 deg; joints [7.088, 56.476, -11.04, -144.326, 51.338, 155.845]
  Set speed (17.9 mm/s)
  Call Extruder(829.98351)
  MoveL 10148 to (533.38, 512.53, 184) mm, rotated rx 180 ry 0 rz 160 deg; joints [7.26, 56.415, -10.925, -144.151, 51.451, 155.76]
  Set speed (17.9 mm/s)
  Call Extruder(834.59366)
  MoveL 10149 to (532.84, 513.88, 184) mm, rotated rx -180 ry 0 rz 160 deg; joints [7.426, 56.344, -10.793, -143.986, 51.569, 155.685]
  Set speed (17.9 mm/s)
  Call Extruder(839.20311)
  MoveL 10150 to (532.24, 515.22, 184) mm, rotated rx -180 ry 0 rz 160 deg; joints [7.591, 56.263, -10.642, -143.826, 51.693, 155.618]
  Set speed (17.9 mm/s)
  Call Extruder(841.50316)
  MoveL 10151 to (531.93, 515.87, 184) mm, rotated rx -180 ry 0 rz 160 deg; joints [7.673, 56.218, -10.559, -143.75, 51.758, 155.588]
  Set speed (17.9 mm/s)
  Call Extruder(844.47065)
  MoveL 10152 to (531.5, 516.71, 184) mm, rotated rx 180 ry 0 rz 160 deg; joints [7.777, 56.157, -10.446, -143.653, 51.844, 155.553]
  Set speed (17.9 mm/s)
  Call Extruder(848.50358)
  MoveL 10153 to (530.88, 517.82, 184) mm, rotated rx -180 ry 0 rz 160 deg; joints [7.918, 56.067, -10.279, -143.526, 51.964, 155.511]
  Set speed (17.8 mm/s)
  Call Extruder(852.21954)
  MoveL 10154 to (530.27, 518.83, 184) mm, rotated rx -180 ry 0 rz 160 deg; joints [8.046, 55.979, -10.114, -143.414, 52.078, 155.477]
  Set speed (17.8 mm/s)
  Call Extruder(855.32986)
  MoveL 10155 to (529.74, 519.66, 184) mm, rotated rx 180 ry 0 rz 160 deg; joints [8.152, 55.899, -9.967, -143.324, 52.177, 155.454]
  Set speed (17.9 mm/s)
  Call Extruder(857.69735)
  MoveL 10156 to (529.32, 520.28, 184) mm, rotated rx -180 ry 0 rz 160 deg; joints [8.231, 55.836, -9.849, -143.257, 52.254, 155.439]
  Set speed (17.9 mm/s)
  Call Extruder(862.30009)
  MoveL 10157 to (528.47, 521.46, 184) mm, rotated rx -180 ry 0 rz 160 deg; joints [8.385, 55.706, -9.607, -143.133, 52.407, 155.416]
  Set speed (17.9 mm/s)
  Call Extruder(864.57871)
  MoveL 10158 to (528.03, 522.03, 184) mm, rotated rx 180 ry 0 rz 160 deg; joints [8.459, 55.638, -9.481, -143.074, 52.484, 155.408]
  Set speed (17.9 mm/s)
  Call Extruder(867.00989)
  MoveL 10159 to (527.55, 522.63, 184) mm, rotated rx 180 ry 0 rz 160 deg; joints [8.538, 55.563, -9.342, -143.013, 52.568, 155.401]
  Call Extruder(869.15314)
  MoveL 10160 to (527.11, 523.15, 184) mm, rotated rx 180 ry 0 rz 160 deg; joints [8.607, 55.495, -9.216, -142.961, 52.644, 155.398]
  Set speed (17.9 mm/s)
  Call Extruder(871.47091)
  MoveL 10161 to (526.63, 523.7, 184) mm, rotated rx 180 ry 0 rz 160 deg; joints [8.681, 55.42, -9.076, -142.907, 52.726, 155.396]
  Call Extruder(873.79285)
  MoveL 10162 to (526.13, 524.25, 184) mm, rotated rx 180 ry 0 rz 160 deg; joints [8.754, 55.343, -8.932, -142.854, 52.809, 155.396]
  Set speed (17.9 mm/s)
  Call Extruder(876.28668)
  MoveL 10163 to (525.59, 524.82, 184) mm, rotated rx 180 ry 0 rz 160 deg; joints [8.831, 55.257, -8.773, -142.799, 52.9, 155.398]
  Set speed (17.9 mm/s)
  Call Extruder(880.80283)
  MoveL 10164 to (524.58, 525.83, 184) mm, rotated rx 180 ry 0 rz 160 deg; joints [8.968, 55.095, -8.473, -142.706, 53.067, 155.409]
  Set speed (17.8 mm/s)
  Call Extruder(883.81779)
  MoveL 10165 to (523.88, 526.48, 184) mm, rotated rx 180 ry 0 rz 160 deg; joints [9.058, 54.984, -8.266, -142.647, 53.181, 155.42]
  Call Extruder(887.67651)
  MoveL 10166 to (522.96, 527.28, 184) mm, rotated rx 180 ry 0 rz 160 deg; joints [9.17, 54.836, -7.991, -142.578, 53.328, 155.44]
  Set speed (17.9 mm/s)
  Call Extruder(889.96561)
